LIN {X 0,Y 456.825,Z 300.941,A -85,B 0,C 180,E1 -8385.675,E2 -8385.675} C_VEL
LIN {X 0,Y 457.17,Z 278.124,A -85,B 0,C 180,E1 -8386.064,E2 -8386.064} C_VEL
LIN {X 0,Y 457.468,Z 213.976,A -85,B 0,C 180,E1 -8387.081,E2 -8387.081} C_VEL
LIN {X 0,Y 453.923,Z 193.615,A -85,B 0,C 180,E1 -8387.574,E2 -8387.574} C_VEL
LIN {X 0,Y 453.952,Z 192.33,A -85,B 0,C 180,E1 -8387.805,E2 -8387.805} C_VEL
LIN {X 0,Y 454.571,Z 180.455,A -85,B 0,C 180,E1 -8390.593,E2 -8390.593} C_VEL
LIN {X 0,Y 455.351,Z 165.331,A -85,B 0,C 180,E1 -8394.045,E2 -8394.045} C_VEL
LIN {X 0,Y 455.413,Z 159.694,A -85,B 0,C 180,E1 -8395.356,E2 -8395.356} C_VEL
LIN {X 0,Y 453.574,Z 149.578,A -85,B 0,C 180,E1 -8397.969,E2 -8397.969} C_VEL
LIN {X 0,Y 453.468,Z 149.499,A -85,B 0,C 180,E1 -8401.525,E2 -8401.525} C_VEL
LIN {X 0,Y 453.488,Z 149.492,A -85,B 0,C 180,E1 -8404.777,E2 -8404.777} C_VEL
LIN {X 0,Y 453.474,Z 149.495,A -85,B 0,C 180,E1 -8408.31,E2 -8408.31} C_VEL
LIN {X 0,Y 453.495,Z 149.481,A -85,B 0,C 180,E1 -8410.608,E2 -8410.608} C_VEL
LIN {X 0,Y 453.455,Z 149.501,A -85,B 0,C 180,E1 -8413.243,E2 -8413.243} C_VEL
LIN {X 0,Y 453.461,Z 149.499,A -85,B 0,C 180,E1 -8415.778,E2 -8415.778} C_VEL
LIN {X 0,Y 453.478,Z 149.495,A -85,B 0,C 180,E1 -8418.209,E2 -8418.209} C_VEL
LIN {X 0,Y 453.486,Z 149.489,A -85,B 0,C 180,E1 -8420.794,E2 -8420.794} C_VEL
LIN {X 0,Y 453.453,Z 149.496,A -85,B 0,C 180,E1 -8423.917,E2 -8423.917} C_VEL
LIN {X 0,Y 453.482,Z 149.491,A -85,B 0,C 180,E1 -8427.151,E2 -8427.151} C_VEL
LIN {X 0,Y 453.473,Z 149.494,A -85,B 0,C 180,E1 -8430.268,E2 -8430.268} C_VEL
LIN {X 0,Y 453.504,Z 149.483,A -85,B 0,C 180,E1 -8433.293,E2 -8433.293} C_VEL
LIN {X 0,Y 453.501,Z 149.49,A -85,B 0,C 180,E1 -8436.238,E2 -8436.238} C_VEL
LIN {X 0,Y 453.48,Z 149.49,A -85,B 0,C 180,E1 -8439.117,E2 -8439.117} C_VEL
LIN {X 0,Y 453.509,Z 149.476,A -85,B 0,C 180,E1 -8441.944,E2 -8441.944} C_VEL
LIN {X 0,Y 453.537,Z 149.489,A -85,B 0,C 180,E1 -8444.726,E2 -8444.726} C_VEL
LIN {X 0,Y 453.556,Z 149.483,A -85,B 0,C 180,E1 -8448.378,E2 -8448.378} C_VEL
LIN {X 0,Y 453.649,Z 149.463,A -85,B 0,C 180,E1 -8451.985,E2 -8451.985} C_VEL
LIN {X 0,Y 453.667,Z 149.476,A -85,B 0,C 180,E1 -8454.666,E2 -8454.666} C_VEL
LIN {X 0,Y 453.741,Z 149.457,A -85,B 0,C 180,E1 -8457.336,E2 -8457.336} C_VEL
LIN {X 0,Y 453.819,Z 149.438,A -85,B 0,C 180,E1 -8460,E2 -8460} C_VEL
LIN {X 0,Y 453.761,Z 149.46,A -85,B 0,C 180,E1 -8462.663,E2 -8462.663} C_VEL
LIN {X 0,Y 453.673,Z 149.474,A -85,B 0,C 180,E1 -8466.225,E2 -8466.225} C_VEL
LIN {X 0,Y 453.588,Z 149.467,A -85,B 0,C 180,E1 -8468.913,E2 -8468.913} C_VEL
LIN {X 0,Y 453.559,Z 149.484,A -85,B 0,C 180,E1 -8472.528,E2 -8472.528} C_VEL
LIN {X 0,Y 453.54,Z 149.486,A -85,B 0,C 180,E1 -8476.196,E2 -8476.196} C_VEL
LIN {X 0,Y 453.515,Z 149.473,A -85,B 0,C 180,E1 -8479.04,E2 -8479.04} C_VEL
LIN {X 0,Y 453.472,Z 149.498,A -85,B 0,C 180,E1 -8481.836,E2 -8481.836} C_VEL
LIN {X 0,Y 453.51,Z 149.489,A -85,B 0,C 180,E1 -8484.734,E2 -8484.734} C_VEL
LIN {X 0,Y 453.532,Z 149.483,A -85,B 0,C 180,E1 -8487.961,E2 -8487.961} C_VEL
LIN {X 0,Y 453.476,Z 149.495,A -85,B 0,C 180,E1 -8490.759,E2 -8490.759} C_VEL
LIN {X 0,Y 453.473,Z 149.486,A -85,B 0,C 180,E1 -8493.912,E2 -8493.912} C_VEL
LIN {X 0,Y 453.465,Z 149.5,A -85,B 0,C 180,E1 -8497.188,E2 -8497.188} C_VEL
LIN {X 0,Y 453.5,Z 149.491,A -85,B 0,C 180,E1 -8499.448,E2 -8499.448} C_VEL
LIN {X 0,Y 453.463,Z 149.5,A -85,B 0,C 180,E1 -8502.994,E2 -8502.994} C_VEL
LIN {X 0,Y 453.467,Z 149.487,A -85,B 0,C 180,E1 -8505.78,E2 -8505.78} C_VEL
LIN {X 0,Y 453.489,Z 149.482,A -85,B 0,C 180,E1 -8509.391,E2 -8509.391} C_VEL
LIN {X 0,Y 453.468,Z 149.497,A -85,B 0,C 180,E1 -8512.223,E2 -8512.223} C_VEL
LIN {X 0,Y 453.484,Z 149.481,A -85,B 0,C 180,E1 -8515.222,E2 -8515.222} C_VEL
LIN {X 0,Y 453.483,Z 149.498,A -85,B 0,C 180,E1 -8518.47,E2 -8518.47} C_VEL
LIN {X 0,Y 453.511,Z 149.487,A -85,B 0,C 180,E1 -8521.289,E2 -8521.289} C_VEL
LIN {X 0,Y 453.52,Z 149.494,A -85,B 0,C 180,E1 -8524.285,E2 -8524.285} C_VEL
LIN {X 0,Y 453.476,Z 149.498,A -85,B 0,C 180,E1 -8527.204,E2 -8527.204} C_VEL
LIN {X 0,Y 453.501,Z 149.496,A -85,B 0,C 180,E1 -8530.066,E2 -8530.066} C_VEL
LIN {X 0,Y 453.503,Z 149.497,A -85,B 0,C 180,E1 -8532.876,E2 -8532.876} C_VEL
LIN {X 0,Y 453.51,Z 149.494,A -85,B 0,C 180,E1 -8535.644,E2 -8535.644} C_VEL
LIN {X 0,Y 453.557,Z 149.491,A -85,B 0,C 180,E1 -8538.379,E2 -8538.379} C_VEL
LIN {X 0,Y 453.648,Z 149.479,A -85,B 0,C 180,E1 -8541.985,E2 -8541.985} C_VEL
LIN {X 0,Y 453.633,Z 149.479,A -85,B 0,C 180,E1 -8543.08,E2 -8543.08} C_VEL
LIN {X 0,Y 452.947,Z 149.567,A -85,B 0,C 180,E1 -8543.82,E2 -8543.82} C_VEL
LIN {X 0,Y 449.998,Z 149.932,A -85,B 0,C 180,E1 -8545.022,E2 -8545.022} C_VEL
LIN {X 0,Y 447.574,Z 150.236,A -85,B 0,C 180,E1 -8545.992,E2 -8545.992} C_VEL
LIN {X 0,Y 446.637,Z 150.352,A -85,B 0,C 180,E1 -8546.742,E2 -8546.742} C_VEL
LIN {X 0,Y 446.617,Z 150.352,A -85,B 0,C 180,E1 -8546.995,E2 -8546.995} C_VEL
LIN {X 0,Y 446.791,Z 150.334,A -85,B 0,C 180,E1 -8550,E2 -8550} C_VEL
LIN {X 0,Y 446.706,Z 150.342,A -85,B 0,C 180,E1 -8552.705,E2 -8552.705} C_VEL
LIN {X 0,Y 446.644,Z 150.351,A -85,B 0,C 180,E1 -8556.324,E2 -8556.324} C_VEL
LIN {X 0,Y 446.535,Z 150.364,A -85,B 0,C 180,E1 -8559.055,E2 -8559.055} C_VEL
LIN {X 0,Y 446.517,Z 150.365,A -85,B 0,C 180,E1 -8562.73,E2 -8562.73} C_VEL
LIN {X 0,Y 446.492,Z 150.369,A -85,B 0,C 180,E1 -8566.228,E2 -8566.228} C_VEL
LIN {X 0,Y 446.466,Z 150.375,A -85,B 0,C 180,E1 -8569.303,E2 -8569.303} C_VEL
LIN {X 0,Y 446.415,Z 150.377,A -85,B 0,C 180,E1 -8572.2,E2 -8572.2} C_VEL
LIN {X 0,Y 446.454,Z 150.376,A -85,B 0,C 180,E1 -8575.152,E2 -8575.152} C_VEL
LIN {X 0,Y 446.48,Z 150.365,A -85,B 0,C 180,E1 -8578.179,E2 -8578.179} C_VEL
LIN {X 0,Y 446.43,Z 150.378,A -85,B 0,C 180,E1 -8581.299,E2 -8581.299} C_VEL
LIN {X 0,Y 446.425,Z 150.36,A -85,B 0,C 180,E1 -8584.523,E2 -8584.523} C_VEL
LIN {X 0,Y 446.426,Z 150.374,A -85,B 0,C 180,E1 -8588.082,E2 -8588.082} C_VEL
LIN {X 0,Y 446.421,Z 150.355,A -85,B 0,C 180,E1 -8590.918,E2 -8590.918} C_VEL
LIN {X 0,Y 446.417,Z 150.363,A -85,B 0,C 180,E1 -8593.843,E2 -8593.843} C_VEL
LIN {X 0,Y 446.416,Z 150.377,A -85,B 0,C 180,E1 -8596.4,E2 -8596.4} C_VEL
LIN {X 0,Y 446.443,Z 150.364,A -85,B 0,C 180,E1 -8599.803,E2 -8599.803} C_VEL
LIN {X 0,Y 446.422,Z 150.376,A -85,B 0,C 180,E1 -8602.123,E2 -8602.123} C_VEL
LIN {X 0,Y 446.425,Z 150.361,A -85,B 0,C 180,E1 -8605.477,E2 -8605.477} C_VEL
LIN {X 0,Y 446.413,Z 150.379,A -85,B 0,C 180,E1 -8608.7,E2 -8608.7} C_VEL
LIN {X 0,Y 446.479,Z 150.362,A -85,B 0,C 180,E1 -8611.822,E2 -8611.822} C_VEL
LIN {X 0,Y 446.454,Z 150.369,A -85,B 0,C 180,E1 -8614.848,E2 -8614.848} C_VEL
LIN {X 0,Y 446.443,Z 150.372,A -85,B 0,C 180,E1 -8618.245,E2 -8618.245} C_VEL
LIN {X 0,Y 446.452,Z 150.355,A -85,B 0,C 180,E1 -8621.65,E2 -8621.65} C_VEL
LIN {X 0,Y 446.503,Z 150.365,A -85,B 0,C 180,E1 -8624.48,E2 -8624.48} C_VEL
LIN {X 0,Y 446.513,Z 150.355,A -85,B 0,C 180,E1 -8628.193,E2 -8628.193} C_VEL
LIN {X 0,Y 446.596,Z 150.345,A -85,B 0,C 180,E1 -8631.858,E2 -8631.858} C_VEL
LIN {X 0,Y 446.641,Z 150.346,A -85,B 0,C 180,E1 -8634.583,E2 -8634.583} C_VEL
LIN {X 0,Y 446.705,Z 150.338,A -85,B 0,C 180,E1 -8637.295,E2 -8637.295} C_VEL
LIN {X 0,Y 446.789,Z 150.313,A -85,B 0,C 180,E1 -8640,E2 -8640} C_VEL
LIN {X 0,Y 446.688,Z 150.336,A -85,B 0,C 180,E1 -8642.706,E2 -8642.706} C_VEL
LIN {X 0,Y 446.643,Z 150.343,A -85,B 0,C 180,E1 -8646.324,E2 -8646.324} C_VEL
LIN {X 0,Y 446.534,Z 150.347,A -85,B 0,C 180,E1 -8649.056,E2 -8649.056} C_VEL
LIN {X 0,Y 446.519,Z 150.358,A -85,B 0,C 180,E1 -8652.73,E2 -8652.73} C_VEL
LIN {X 0,Y 446.494,Z 150.359,A -85,B 0,C 180,E1 -8656.228,E2 -8656.228} C_VEL
LIN {X 0,Y 446.467,Z 150.357,A -85,B 0,C 180,E1 -8659.304,E2 -8659.304} C_VEL
LIN {X 0,Y 446.416,Z 150.372,A -85,B 0,C 180,E1 -8662.2,E2 -8662.2} C_VEL
LIN {X 0,Y 446.455,Z 150.365,A -85,B 0,C 180,E1 -8665.153,E2 -8665.153} C_VEL
LIN {X 0,Y 446.483,Z 150.357,A -85,B 0,C 180,E1 -8668.179,E2 -8668.179} C_VEL
LIN {X 0,Y 446.418,Z 150.373,A -85,B 0,C 180,E1 -8671.776,E2 -8671.776} C_VEL
LIN {X 0,Y 446.428,Z 150.366,A -85,B 0,C 180,E1 -8674.524,E2 -8674.524} C_VEL
LIN {X 0,Y 446.412,Z 150.377,A -85,B 0,C 180,E1 -8678.079,E2 -8678.079} C_VEL
LIN {X 0,Y 446.426,Z 150.375,A -85,B 0,C 180,E1 -8680.918,E2 -8680.918} C_VEL
LIN {X 0,Y 446.397,Z 150.377,A -85,B 0,C 180,E1 -8683.847,E2 -8683.847} C_VEL
LIN {X 0,Y 446.398,Z 150.383,A -85,B 0,C 180,E1 -8686.404,E2 -8686.404} C_VEL
LIN {X 0,Y 446.427,Z 150.361,A -85,B 0,C 180,E1 -8689.083,E2 -8689.083} C_VEL
LIN {X 0,Y 446.428,Z 150.377,A -85,B 0,C 180,E1 -8692.124,E2 -8692.124} C_VEL
LIN {X 0,Y 446.43,Z 150.371,A -85,B 0,C 180,E1 -8695.477,E2 -8695.477} C_VEL
LIN {X 0,Y 446.418,Z 150.38,A -85,B 0,C 180,E1 -8698.7,E2 -8698.7} C_VEL
LIN {X 0,Y 446.522,Z 150.503,A -85,B 0,C 180,E1 -8701.824,E2 -8701.824} C_VEL
LIN {X 0,Y 448.185,Z 159.571,A -85,B 0,C 180,E1 -8704.206,E2 -8704.206} C_VEL
LIN {X 0,Y 448.462,Z 164.125,A -85,B 0,C 180,E1 -8705.36,E2 -8705.36} C_VEL
LIN {X 0,Y 447.654,Z 179.053,A -85,B 0,C 180,E1 -8708.833,E2 -8708.833} C_VEL
LIN {X 0,Y 446.966,Z 192.145,A -85,B 0,C 180,E1 -8711.908,E2 -8711.908} C_VEL
LIN {X 0,Y 446.955,Z 193.46,A -85,B 0,C 180,E1 -8712.145,E2 -8712.145} C_VEL
LIN {X 0,Y 450.797,Z 215.824,A -85,B 0,C 180,E1 -8712.691,E2 -8712.691} C_VEL
LIN {X 0,Y 450.061,Z 298.086,A -85,B 0,C 180,E1 -8714.025,E2 -8714.025} C_VEL
LIN {X 0,Y 449.811,Z 307.982,A -85,B 0,C 180,E1 -8714.277,E2 -8714.277} C_VEL
LIN {X 0,Y 449.447,Z 317.957,A -85,B 0,C 180,E1 -8714.642,E2 -8714.642} C_VEL
LIN {X 0,Y 449.065,Z 327.314,A -85,B 0,C 180,E1 -8715.093,E2 -8715.093} C_VEL
LIN {X 0,Y 448.597,Z 335.823,A -85,B 0,C 180,E1 -8715.599,E2 -8715.599} C_VEL
LIN {X 0,Y 448.084,Z 345.1,A -85,B 0,C 180,E1 -8716.277,E2 -8716.277} C_VEL
LIN {X 0,Y 447.67,Z 353.812,A -85,B 0,C 180,E1 -8717.049,E2 -8717.049} C_VEL
LIN {X 0,Y 447.137,Z 362.58,A -85,B 0,C 180,E1 -8717.98,E2 -8717.98} C_VEL
LIN {X 0,Y 446.696,Z 369.8,A -85,B 0,C 180,E1 -8718.888,E2 -8718.888} C_VEL
LIN {X 0,Y 446.358,Z 376.003,A -85,B 0,C 180,E1 -8719.797,E2 -8719.797} C_VEL
LIN {X 0,Y 445.997,Z 382.54,A -85,B 0,C 180,E1 -8720.934,E2 -8720.934} C_VEL
LIN {X 0,Y 445.785,Z 387.041,A -85,B 0,C 180,E1 -8721.843,E2 -8721.843} C_VEL
LIN {X 0,Y 445.57,Z 392.533,A -85,B 0,C 180,E1 -8723.207,E2 -8723.207} C_VEL
LIN {X 0,Y 445.476,Z 396.854,A -85,B 0,C 180,E1 -8724.568,E2 -8724.568} C_VEL
LIN {X 0,Y 445.413,Z 399.219,A -85,B 0,C 180,E1 -8725.475,E2 -8725.475} C_VEL
LIN {X 0,Y 445.433,Z 402.402,A -85,B 0,C 180,E1 -8727.287,E2 -8727.287} C_VEL
LIN {X 0,Y 445.356,Z 403.457,A -85,B 0,C 180,E1 -8728.191,E2 -8728.191} C_VEL
LIN {X 0,Y 445.34,Z 404.044,A -85,B 0,C 180,E1 -8729.096,E2 -8729.096} C_VEL
LIN {X 0,Y 445.34,Z 404.044,A -85,B 0,C 180,E1 -8730.904,E2 -8730.904} C_VEL
LIN {X 0,Y 445.356,Z 403.457,A -85,B 0,C 180,E1 -8731.809,E2 -8731.809} C_VEL
LIN {X 0,Y 445.433,Z 402.402,A -85,B 0,C 180,E1 -8732.713,E2 -8732.713} C_VEL
LIN {X 0,Y 445.413,Z 399.219,A -85,B 0,C 180,E1 -8734.525,E2 -8734.525} C_VEL
LIN {X 0,Y 445.469,Z 395.105,A -85,B 0,C 180,E1 -8736.041,E2 -8736.041} C_VEL
LIN {X 0,Y 445.601,Z 390.871,A -85,B 0,C 180,E1 -8737.249,E2 -8737.249} C_VEL
LIN {X 0,Y 445.889,Z 384.851,A -85,B 0,C 180,E1 -8738.612,E2 -8738.612} C_VEL
LIN {X 0,Y 446.194,Z 378.755,A -85,B 0,C 180,E1 -8739.748,E2 -8739.748} C_VEL
LIN {X 0,Y 446.498,Z 373.054,A -85,B 0,C 180,E1 -8740.658,E2 -8740.658} C_VEL
LIN {X 0,Y 447.04,Z 364.5,A -85,B 0,C 180,E1 -8741.793,E2 -8741.793} C_VEL
LIN {X 0,Y 447.502,Z 356.319,A -85,B 0,C 180,E1 -8742.701,E2 -8742.701} C_VEL
LIN {X 0,Y 447.957,Z 347.932,A -85,B 0,C 180,E1 -8743.485,E2 -8743.485} C_VEL
LIN {X 0,Y 448.42,Z 339.087,A -85,B 0,C 180,E1 -8744.175,E2 -8744.175} C_VEL
LIN {X 0,Y 448.916,Z 329.327,A -85,B 0,C 180,E1 -8744.796,E2 -8744.796} C_VEL
LIN {X 0,Y 449.344,Z 320.533,A -85,B 0,C 180,E1 -8745.245,E2 -8745.245} C_VEL
LIN {X 0,Y 449.727,Z 310.605,A -85,B 0,C 180,E1 -8745.639,E2 -8745.639} C_VEL
LIN {X 0,Y 450.008,Z 300.75,A -85,B 0,C 180,E1 -8745.919,E2 -8745.919} C_VEL
LIN {X 0,Y 450.402,Z 275.651,A -85,B 0,C 180,E1 -8746.349,E2 -8746.349} C_VEL
LIN {X 0,Y 450.678,Z 214.695,A -85,B 0,C 180,E1 -8747.332,E2 -8747.332} C_VEL
LIN {X 0,Y 446.964,Z 193.579,A -85,B 0,C 180,E1 -8747.846,E2 -8747.846} C_VEL
LIN {X 0,Y 446.931,Z 192.787,A -85,B 0,C 180,E1 -8747.942,E2 -8747.942} C_VEL
LIN {X 0,Y 447.636,Z 180.293,A -85,B 0,C 180,E1 -8750.927,E2 -8750.927} C_VEL
LIN {X 0,Y 448.451,Z 165.578,A -85,B 0,C 180,E1 -8754.349,E2 -8754.349} C_VEL
LIN {X 0,Y 448.395,Z 160.582,A -85,B 0,C 180,E1 -8755.532,E2 -8755.532} C_VEL
LIN {X 0,Y 446.524,Z 150.482,A -85,B 0,C 180,E1 -8758.187,E2 -8758.187} C_VEL
LIN {X 0,Y 446.421,Z 150.374,A -85,B 0,C 180,E1 -8761.774,E2 -8761.774} C_VEL
LIN {X 0,Y 446.43,Z 150.372,A -85,B 0,C 180,E1 -8764.523,E2 -8764.523} C_VEL
LIN {X 0,Y 446.431,Z 150.375,A -85,B 0,C 180,E1 -8768.081,E2 -8768.081} C_VEL
LIN {X 0,Y 446.427,Z 150.361,A -85,B 0,C 180,E1 -8770.917,E2 -8770.917} C_VEL
LIN {X 0,Y 446.4,Z 150.379,A -85,B 0,C 180,E1 -8773.846,E2 -8773.846} C_VEL
LIN {X 0,Y 446.396,Z 150.377,A -85,B 0,C 180,E1 -8776.403,E2 -8776.403} C_VEL
LIN {X 0,Y 446.426,Z 150.375,A -85,B 0,C 180,E1 -8779.082,E2 -8779.082} C_VEL
LIN {X 0,Y 446.406,Z 150.376,A -85,B 0,C 180,E1 -8782.12,E2 -8782.12} C_VEL
LIN {X 0,Y 446.428,Z 150.366,A -85,B 0,C 180,E1 -8785.476,E2 -8785.476} C_VEL
LIN {X 0,Y 446.415,Z 150.375,A -85,B 0,C 180,E1 -8788.699,E2 -8788.699} C_VEL
LIN {X 0,Y 446.483,Z 150.357,A -85,B 0,C 180,E1 -8791.821,E2 -8791.821} C_VEL
LIN {X 0,Y 446.455,Z 150.365,A -85,B 0,C 180,E1 -8794.847,E2 -8794.847} C_VEL
LIN {X 0,Y 446.446,Z 150.369,A -85,B 0,C 180,E1 -8798.245,E2 -8798.245} C_VEL
LIN {X 0,Y 446.454,Z 150.354,A -85,B 0,C 180,E1 -8801.649,E2 -8801.649} C_VEL
LIN {X 0,Y 446.505,Z 150.362,A -85,B 0,C 180,E1 -8804.479,E2 -8804.479} C_VEL
LIN {X 0,Y 446.514,Z 150.359,A -85,B 0,C 180,E1 -8808.193,E2 -8808.193} C_VEL
LIN {X 0,Y 446.597,Z 150.34,A -85,B 0,C 180,E1 -8811.857,E2 -8811.857} C_VEL
LIN {X 0,Y 446.642,Z 150.352,A -85,B 0,C 180,E1 -8814.582,E2 -8814.582} C_VEL
LIN {X 0,Y 446.66,Z 150.34,A -85,B 0,C 180,E1 -8818.196,E2 -8818.196} C_VEL
LIN {X 0,Y 446.789,Z 150.313,A -85,B 0,C 180,E1 -8820,E2 -8820} C_VEL
LIN {X 0,Y 446.705,Z 150.338,A -85,B 0,C 180,E1 -8822.705,E2 -8822.705} C_VEL
LIN {X 0,Y 446.642,Z 150.348,A -85,B 0,C 180,E1 -8826.323,E2 -8826.323} C_VEL
LIN {X 0,Y 446.534,Z 150.344,A -85,B 0,C 180,E1 -8829.055,E2 -8829.055} C_VEL
LIN {X 0,Y 446.517,Z 150.36,A -85,B 0,C 180,E1 -8832.729,E2 -8832.729} C_VEL
LIN {X 0,Y 446.492,Z 150.364,A -85,B 0,C 180,E1 -8836.228,E2 -8836.228} C_VEL
LIN {X 0,Y 446.464,Z 150.352,A -85,B 0,C 180,E1 -8839.303,E2 -8839.303} C_VEL
LIN {X 0,Y 446.414,Z 150.377,A -85,B 0,C 180,E1 -8842.199,E2 -8842.199} C_VEL
LIN {X 0,Y 446.454,Z 150.369,A -85,B 0,C 180,E1 -8845.152,E2 -8845.152} C_VEL
LIN {X 0,Y 446.479,Z 150.362,A -85,B 0,C 180,E1 -8848.178,E2 -8848.178} C_VEL
LIN {X 0,Y 446.413,Z 150.379,A -85,B 0,C 180,E1 -8851.3,E2 -8851.3} C_VEL
LIN {X 0,Y 446.425,Z 150.361,A -85,B 0,C 180,E1 -8854.523,E2 -8854.523} C_VEL
LIN {X 0,Y 446.425,Z 150.374,A -85,B 0,C 180,E1 -8858.082,E2 -8858.082} C_VEL
LIN {X 0,Y 446.422,Z 150.368,A -85,B 0,C 180,E1 -8860.918,E2 -8860.918} C_VEL
LIN {X 0,Y 446.418,Z 150.374,A -85,B 0,C 180,E1 -8863.843,E2 -8863.843} C_VEL
LIN {X 0,Y 446.415,Z 150.364,A -85,B 0,C 180,E1 -8866.4,E2 -8866.4} C_VEL
LIN {X 0,Y 446.438,Z 150.366,A -85,B 0,C 180,E1 -8869.802,E2 -8869.802} C_VEL
LIN {X 0,Y 446.423,Z 150.375,A -85,B 0,C 180,E1 -8872.123,E2 -8872.123} C_VEL
LIN {X 0,Y 446.426,Z 150.36,A -85,B 0,C 180,E1 -8875.477,E2 -8875.477} C_VEL
LIN {X 0,Y 446.43,Z 150.378,A -85,B 0,C 180,E1 -8878.701,E2 -8878.701} C_VEL
LIN {X 0,Y 446.48,Z 150.365,A -85,B 0,C 180,E1 -8881.821,E2 -8881.821} C_VEL
LIN {X 0,Y 446.454,Z 150.376,A -85,B 0,C 180,E1 -8884.848,E2 -8884.848} C_VEL
LIN {X 0,Y 446.444,Z 150.376,A -85,B 0,C 180,E1 -8888.245,E2 -8888.245} C_VEL
LIN {X 0,Y 446.454,Z 150.373,A -85,B 0,C 180,E1 -8891.649,E2 -8891.649} C_VEL
LIN {X 0,Y 446.504,Z 150.37,A -85,B 0,C 180,E1 -8894.48,E2 -8894.48} C_VEL
LIN {X 0,Y 446.514,Z 150.368,A -85,B 0,C 180,E1 -8898.193,E2 -8898.193} C_VEL
LIN {X 0,Y 446.597,Z 150.357,A -85,B 0,C 180,E1 -8901.858,E2 -8901.858} C_VEL
LIN {X 0,Y 446.643,Z 150.351,A -85,B 0,C 180,E1 -8904.583,E2 -8904.583} C_VEL
LIN {X 0,Y 446.617,Z 150.352,A -85,B 0,C 180,E1 -8906.995,E2 -8906.995} C_VEL
LIN {X 0,Y 446.1,Z 150.42,A -85,B 0,C 180,E1 -8907.748,E2 -8907.748} C_VEL
LIN {X 0,Y 443.286,Z 150.772,A -85,B 0,C 180,E1 -8908.971,E2 -8908.971} C_VEL
LIN {X 0,Y 440.802,Z 151.081,A -85,B 0,C 180,E1 -8909.958,E2 -8909.958} C_VEL
LIN {X 0,Y 439.713,Z 151.214,A -85,B 0,C 180,E1 -8910.721,E2 -8910.721} C_VEL
LIN {X 0,Y 439.619,Z 151.225,A -85,B 0,C 180,E1 -8910.98,E2 -8910.98} C_VEL
LIN {X 0,Y 439.653,Z 151.221,A -85,B 0,C 180,E1 -8912.749,E2 -8912.749} C_VEL
LIN {X 0,Y 439.615,Z 151.226,A -85,B 0,C 180,E1 -8916.425,E2 -8916.425} C_VEL
LIN {X 0,Y 439.497,Z 151.241,A -85,B 0,C 180,E1 -8919.202,E2 -8919.202} C_VEL
LIN {X 0,Y 439.462,Z 151.245,A -85,B 0,C 180,E1 -8922.938,E2 -8922.938} C_VEL
LIN {X 0,Y 439.444,Z 151.246,A -85,B 0,C 180,E1 -8926.349,E2 -8926.349} C_VEL
LIN {X 0,Y 439.399,Z 151.255,A -85,B 0,C 180,E1 -8929.626,E2 -8929.626} C_VEL
LIN {X 0,Y 439.362,Z 151.256,A -85,B 0,C 180,E1 -8932.575,E2 -8932.575} C_VEL
LIN {X 0,Y 439.401,Z 151.254,A -85,B 0,C 180,E1 -8935.585,E2 -8935.585} C_VEL
LIN {X 0,Y 439.421,Z 151.241,A -85,B 0,C 180,E1 -8938.673,E2 -8938.673} C_VEL
LIN {X 0,Y 439.381,Z 151.252,A -85,B 0,C 180,E1 -8942.034,E2 -8942.034} C_VEL
LIN {X 0,Y 439.391,Z 151.239,A -85,B 0,C 180,E1 -8945.341,E2 -8945.341} C_VEL
LIN {X 0,Y 439.379,Z 151.255,A -85,B 0,C 180,E1 -8948.595,E2 -8948.595} C_VEL
LIN {X 0,Y 439.383,Z 151.226,A -85,B 0,C 180,E1 -8951.257,E2 -8951.257} C_VEL
LIN {X 0,Y 439.401,Z 151.243,A -85,B 0,C 180,E1 -8954.729,E2 -8954.729} C_VEL
LIN {X 0,Y 439.393,Z 151.248,A -85,B 0,C 180,E1 -8957.796,E2 -8957.796} C_VEL
LIN {X 0,Y 439.425,Z 151.24,A -85,B 0,C 180,E1 -8960.228,E2 -8960.228} C_VEL
LIN {X 0,Y 439.372,Z 151.251,A -85,B 0,C 180,E1 -8963.713,E2 -8963.713} C_VEL
LIN {X 0,Y 439.368,Z 151.252,A -85,B 0,C 180,E1 -8967.054,E2 -8967.054} C_VEL
LIN {X 0,Y 439.386,Z 151.254,A -85,B 0,C 180,E1 -8970.275,E2 -8970.275} C_VEL
LIN {X 0,Y 439.425,Z 151.234,A -85,B 0,C 180,E1 -8973.397,E2 -8973.397} C_VEL
LIN {X 0,Y 439.383,Z 151.255,A -85,B 0,C 180,E1 -8976.43,E2 -8976.43} C_VEL
LIN {X 0,Y 439.383,Z 151.244,A -85,B 0,C 180,E1 -8979.397,E2 -8979.397} C_VEL
LIN {X 0,Y 439.427,Z 151.239,A -85,B 0,C 180,E1 -8982.31,E2 -8982.31} C_VEL
LIN {X 0,Y 439.443,Z 151.243,A -85,B 0,C 180,E1 -8985.174,E2 -8985.174} C_VEL
LIN {X 0,Y 439.479,Z 151.233,A -85,B 0,C 180,E1 -8988.002,E2 -8988.002} C_VEL
LIN {X 0,Y 439.544,Z 151.221,A -85,B 0,C 180,E1 -8991.727,E2 -8991.727} C_VEL
LIN {X 0,Y 439.617,Z 151.221,A -85,B 0,C 180,E1 -8994.496,E2 -8994.496} C_VEL
LIN {X 0,Y 439.632,Z 151.208,A -85,B 0,C 180,E1 -8998.168,E2 -8998.168} C_VEL
LIN {X 0,Y 439.758,Z 151.188,A -85,B 0,C 180,E1 -9000,E2 -9000} C_VEL
LIN {X 0,Y 439.638,Z 151.214,A -85,B 0,C 180,E1 -9002.749,E2 -9002.749} C_VEL
LIN {X 0,Y 439.615,Z 151.219,A -85,B 0,C 180,E1 -9006.426,E2 -9006.426} C_VEL
LIN {X 0,Y 439.496,Z 151.222,A -85,B 0,C 180,E1 -9009.202,E2 -9009.202} C_VEL
LIN {X 0,Y 439.463,Z 151.238,A -85,B 0,C 180,E1 -9012.938,E2 -9012.938} C_VEL
LIN {X 0,Y 439.445,Z 151.238,A -85,B 0,C 180,E1 -9016.349,E2 -9016.349} C_VEL
LIN {X 0,Y 439.4,Z 151.24,A -85,B 0,C 180,E1 -9019.627,E2 -9019.627} C_VEL
LIN {X 0,Y 439.363,Z 151.253,A -85,B 0,C 180,E1 -9022.576,E2 -9022.576} C_VEL
LIN {X 0,Y 439.403,Z 151.239,A -85,B 0,C 180,E1 -9025.585,E2 -9025.585} C_VEL
LIN {X 0,Y 439.416,Z 151.242,A -85,B 0,C 180,E1 -9028.674,E2 -9028.674} C_VEL
LIN {X 0,Y 439.369,Z 151.251,A -85,B 0,C 180,E1 -9032.031,E2 -9032.031} C_VEL
LIN {X 0,Y 439.393,Z 151.246,A -85,B 0,C 180,E1 -9035.341,E2 -9035.341} C_VEL
LIN {X 0,Y 439.374,Z 151.253,A -85,B 0,C 180,E1 -9038.596,E2 -9038.596} C_VEL
LIN {X 0,Y 439.388,Z 151.249,A -85,B 0,C 180,E1 -9041.257,E2 -9041.257} C_VEL
LIN {X 0,Y 439.399,Z 151.249,A -85,B 0,C 180,E1 -9044.73,E2 -9044.73} C_VEL
LIN {X 0,Y 439.396,Z 151.25,A -85,B 0,C 180,E1 -9047.796,E2 -9047.796} C_VEL
LIN {X 0,Y 439.43,Z 151.234,A -85,B 0,C 180,E1 -9050.228,E2 -9050.228} C_VEL
LIN {X 0,Y 439.375,Z 151.251,A -85,B 0,C 180,E1 -9053.713,E2 -9053.713} C_VEL
LIN {X 0,Y 439.374,Z 151.252,A -85,B 0,C 180,E1 -9057.055,E2 -9057.055} C_VEL
LIN {X 0,Y 439.384,Z 151.25,A -85,B 0,C 180,E1 -9060.275,E2 -9060.275} C_VEL
LIN {X 0,Y 439.476,Z 151.376,A -85,B 0,C 180,E1 -9061.589,E2 -9061.589} C_VEL
LIN {X 0,Y 441.152,Z 160.441,A -85,B 0,C 180,E1 -9064.017,E2 -9064.017} C_VEL
LIN {X 0,Y 441.533,Z 164.726,A -85,B 0,C 180,E1 -9065.133,E2 -9065.133} C_VEL
LIN {X 0,Y 440.669,Z 179.922,A -85,B 0,C 180,E1 -9068.726,E2 -9068.726} C_VEL
LIN {X 0,Y 439.998,Z 191.956,A -85,B 0,C 180,E1 -9071.612,E2 -9071.612} C_VEL
LIN {X 0,Y 439.991,Z 193.272,A -85,B 0,C 180,E1 -9071.853,E2 -9071.853} C_VEL
LIN {X 0,Y 444.019,Z 216.881,A -85,B 0,C 180,E1 -9072.439,E2 -9072.439} C_VEL
LIN {X 0,Y 443.239,Z 297.895,A -85,B 0,C 180,E1 -9073.772,E2 -9073.772} C_VEL
LIN {X 0,Y 442.974,Z 307.79,A -85,B 0,C 180,E1 -9074.028,E2 -9074.028} C_VEL
LIN {X 0,Y 442.615,Z 317.766,A -85,B 0,C 180,E1 -9074.399,E2 -9074.399} C_VEL
LIN {X 0,Y 442.152,Z 328.13,A -85,B 0,C 180,E1 -9074.913,E2 -9074.913} C_VEL
LIN {X 0,Y 441.617,Z 337.263,A -85,B 0,C 180,E1 -9075.484,E2 -9075.484} C_VEL
LIN {X 0,Y 441.101,Z 346.261,A -85,B 0,C 180,E1 -9076.173,E2 -9076.173} C_VEL
LIN {X 0,Y 440.676,Z 354.409,A -85,B 0,C 180,E1 -9076.921,E2 -9076.921} C_VEL
LIN {X 0,Y 440.177,Z 362.388,A -85,B 0,C 180,E1 -9077.787,E2 -9077.787} C_VEL
LIN {X 0,Y 439.712,Z 369.608,A -85,B 0,C 180,E1 -9078.709,E2 -9078.709} C_VEL
LIN {X 0,Y 439.342,Z 375.81,A -85,B 0,C 180,E1 -9079.633,E2 -9079.633} C_VEL
LIN {X 0,Y 438.97,Z 382.348,A -85,B 0,C 180,E1 -9080.787,E2 -9080.787} C_VEL
LIN {X 0,Y 438.739,Z 386.849,A -85,B 0,C 180,E1 -9081.711,E2 -9081.711} C_VEL
LIN {X 0,Y 438.499,Z 392.339,A -85,B 0,C 180,E1 -9083.096,E2 -9083.096} C_VEL
LIN {X 0,Y 438.374,Z 396.662,A -85,B 0,C 180,E1 -9084.48,E2 -9084.48} C_VEL
LIN {X 0,Y 438.342,Z 399.027,A -85,B 0,C 180,E1 -9085.402,E2 -9085.402} C_VEL
LIN {X 0,Y 438.341,Z 402.211,A -85,B 0,C 180,E1 -9087.243,E2 -9087.243} C_VEL
LIN {X 0,Y 438.279,Z 403.266,A -85,B 0,C 180,E1 -9088.162,E2 -9088.162} C_VEL
LIN {X 0,Y 438.253,Z 403.853,A -85,B 0,C 180,E1 -9089.081,E2 -9089.081} C_VEL
LIN {X 0,Y 438.253,Z 403.853,A -85,B 0,C 180,E1 -9090.919,E2 -9090.919} C_VEL
LIN {X 0,Y 438.279,Z 403.266,A -85,B 0,C 180,E1 -9091.838,E2 -9091.838} C_VEL
LIN {X 0,Y 438.341,Z 402.211,A -85,B 0,C 180,E1 -9092.757,E2 -9092.757} C_VEL
LIN {X 0,Y 438.342,Z 399.027,A -85,B 0,C 180,E1 -9094.598,E2 -9094.598} C_VEL
LIN {X 0,Y 438.423,Z 394.227,A -85,B 0,C 180,E1 -9096.343,E2 -9096.343} C_VEL
LIN {X 0,Y 438.633,Z 388.764,A -85,B 0,C 180,E1 -9097.827,E2 -9097.827} C_VEL
LIN {X 0,Y 438.891,Z 383.503,A -85,B 0,C 180,E1 -9098.982,E2 -9098.982} C_VEL
LIN {X 0,Y 439.247,Z 377.186,A -85,B 0,C 180,E1 -9100.137,E2 -9100.137} C_VEL
LIN {X 0,Y 439.582,Z 371.234,A -85,B 0,C 180,E1 -9101.061,E2 -9101.061} C_VEL
LIN {X 0,Y 440.063,Z 364.307,A -85,B 0,C 180,E1 -9101.983,E2 -9101.983} C_VEL
LIN {X 0,Y 440.54,Z 356.126,A -85,B 0,C 180,E1 -9102.905,E2 -9102.905} C_VEL
LIN {X 0,Y 441.009,Z 348.189,A -85,B 0,C 180,E1 -9103.662,E2 -9103.662} C_VEL
LIN {X 0,Y 441.532,Z 338.895,A -85,B 0,C 180,E1 -9104.401,E2 -9104.401} C_VEL
LIN {X 0,Y 442.041,Z 329.135,A -85,B 0,C 180,E1 -9105.031,E2 -9105.031} C_VEL
LIN {X 0,Y 442.599,Z 319.055,A -85,B 0,C 180,E1 -9105.543,E2 -9105.543} C_VEL
LIN {X 0,Y 442.921,Z 309.539,A -85,B 0,C 180,E1 -9105.915,E2 -9105.915} C_VEL
LIN {X 0,Y 443.2,Z 300.559,A -85,B 0,C 180,E1 -9106.17,E2 -9106.17} C_VEL
LIN {X 0,Y 443.601,Z 275.568,A -85,B 0,C 180,E1 -9106.605,E2 -9106.605} C_VEL
LIN {X 0,Y 443.964,Z 215.957,A -85,B 0,C 180,E1 -9107.578,E2 -9107.578} C_VEL
LIN {X 0,Y 439.969,Z 193.239,A -85,B 0,C 180,E1 -9108.15,E2 -9108.15} C_VEL
LIN {X 0,Y 439.983,Z 192.049,A -85,B 0,C 180,E1 -9108.365,E2 -9108.365} C_VEL
LIN {X 0,Y 440.674,Z 180.13,A -85,B 0,C 180,E1 -9111.273,E2 -9111.273} C_VEL
LIN {X 0,Y 441.489,Z 166.736,A -85,B 0,C 180,E1 -9114.449,E2 -9114.449} C_VEL
LIN {X 0,Y 441.527,Z 162.54,A -85,B 0,C 180,E1 -9115.453,E2 -9115.453} C_VEL
LIN {X 0,Y 439.75,Z 152.83,A -85,B 0,C 180,E1 -9118.001,E2 -9118.001} C_VEL
LIN {X 0,Y 439.446,Z 151.268,A -85,B 0,C 180,E1 -9118.493,E2 -9118.493} C_VEL
LIN {X 0,Y 439.372,Z 151.251,A -85,B 0,C 180,E1 -9122.03,E2 -9122.03} C_VEL
LIN {X 0,Y 439.395,Z 151.244,A -85,B 0,C 180,E1 -9125.34,E2 -9125.34} C_VEL
LIN {X 0,Y 439.389,Z 151.248,A -85,B 0,C 180,E1 -9128.594,E2 -9128.594} C_VEL
LIN {X 0,Y 439.389,Z 151.24,A -85,B 0,C 180,E1 -9131.256,E2 -9131.256} C_VEL
LIN {X 0,Y 439.399,Z 151.247,A -85,B 0,C 180,E1 -9134.729,E2 -9134.729} C_VEL
LIN {X 0,Y 439.395,Z 151.252,A -85,B 0,C 180,E1 -9137.795,E2 -9137.795} C_VEL
LIN {X 0,Y 439.394,Z 151.243,A -85,B 0,C 180,E1 -9140.223,E2 -9140.223} C_VEL
LIN {X 0,Y 439.373,Z 151.251,A -85,B 0,C 180,E1 -9143.712,E2 -9143.712} C_VEL
LIN {X 0,Y 439.371,Z 151.247,A -85,B 0,C 180,E1 -9147.053,E2 -9147.053} C_VEL
LIN {X 0,Y 439.381,Z 151.25,A -85,B 0,C 180,E1 -9150.274,E2 -9150.274} C_VEL
LIN {X 0,Y 439.427,Z 151.236,A -85,B 0,C 180,E1 -9153.396,E2 -9153.396} C_VEL
LIN {X 0,Y 439.384,Z 151.249,A -85,B 0,C 180,E1 -9156.429,E2 -9156.429} C_VEL
LIN {X 0,Y 439.386,Z 151.242,A -85,B 0,C 180,E1 -9159.396,E2 -9159.396} C_VEL
LIN {X 0,Y 439.429,Z 151.23,A -85,B 0,C 180,E1 -9162.309,E2 -9162.309} C_VEL
LIN {X 0,Y 439.446,Z 151.244,A -85,B 0,C 180,E1 -9165.173,E2 -9165.173} C_VEL
LIN {X 0,Y 439.48,Z 151.233,A -85,B 0,C 180,E1 -9168.001,E2 -9168.001} C_VEL
LIN {X 0,Y 439.545,Z 151.218,A -85,B 0,C 180,E1 -9171.726,E2 -9171.726} C_VEL
LIN {X 0,Y 439.618,Z 151.226,A -85,B 0,C 180,E1 -9174.495,E2 -9174.495} C_VEL
LIN {X 0,Y 439.63,Z 151.216,A -85,B 0,C 180,E1 -9178.167,E2 -9178.167} C_VEL
LIN {X 0,Y 439.758,Z 151.188,A -85,B 0,C 180,E1 -9180,E2 -9180} C_VEL
LIN {X 0,Y 439.652,Z 151.216,A -85,B 0,C 180,E1 -9182.748,E2 -9182.748} C_VEL
LIN {X 0,Y 439.614,Z 151.222,A -85,B 0,C 180,E1 -9186.425,E2 -9186.425} C_VEL
LIN {X 0,Y 439.496,Z 151.221,A -85,B 0,C 180,E1 -9189.201,E2 -9189.201} C_VEL
LIN {X 0,Y 439.461,Z 151.238,A -85,B 0,C 180,E1 -9192.937,E2 -9192.937} C_VEL
LIN {X 0,Y 439.443,Z 151.24,A -85,B 0,C 180,E1 -9196.348,E2 -9196.348} C_VEL
LIN {X 0,Y 439.398,Z 151.234,A -85,B 0,C 180,E1 -9199.626,E2 -9199.626} C_VEL
LIN {X 0,Y 439.361,Z 151.253,A -85,B 0,C 180,E1 -9202.575,E2 -9202.575} C_VEL
LIN {X 0,Y 439.401,Z 151.246,A -85,B 0,C 180,E1 -9205.584,E2 -9205.584} C_VEL
LIN {X 0,Y 439.416,Z 151.24,A -85,B 0,C 180,E1 -9208.673,E2 -9208.673} C_VEL
LIN {X 0,Y 439.369,Z 151.254,A -85,B 0,C 180,E1 -9211.86,E2 -9211.86} C_VEL
LIN {X 0,Y 439.396,Z 151.24,A -85,B 0,C 180,E1 -9215.156,E2 -9215.156} C_VEL
LIN {X 0,Y 439.383,Z 151.251,A -85,B 0,C 180,E1 -9218.594,E2 -9218.594} C_VEL
LIN {X 0,Y 439.384,Z 151.247,A -85,B 0,C 180,E1 -9221.257,E2 -9221.257} C_VEL
LIN {X 0,Y 439.401,Z 151.25,A -85,B 0,C 180,E1 -9224.728,E2 -9224.728} C_VEL
LIN {X 0,Y 439.391,Z 151.221,A -85,B 0,C 180,E1 -9227.796,E2 -9227.796} C_VEL
LIN {X 0,Y 439.421,Z 151.24,A -85,B 0,C 180,E1 -9230.227,E2 -9230.227} C_VEL
LIN {X 0,Y 439.372,Z 151.247,A -85,B 0,C 180,E1 -9233.713,E2 -9233.713} C_VEL
LIN {X 0,Y 439.372,Z 151.251,A -85,B 0,C 180,E1 -9237.054,E2 -9237.054} C_VEL
LIN {X 0,Y 439.393,Z 151.243,A -85,B 0,C 180,E1 -9240.275,E2 -9240.275} C_VEL
LIN {X 0,Y 439.429,Z 151.247,A -85,B 0,C 180,E1 -9243.589,E2 -9243.589} C_VEL
LIN {X 0,Y 439.383,Z 151.257,A -85,B 0,C 180,E1 -9246.43,E2 -9246.43} C_VEL
LIN {X 0,Y 439.385,Z 151.253,A -85,B 0,C 180,E1 -9249.397,E2 -9249.397} C_VEL
LIN {X 0,Y 439.428,Z 151.251,A -85,B 0,C 180,E1 -9252.31,E2 -9252.31} C_VEL
LIN {X 0,Y 439.444,Z 151.247,A -85,B 0,C 180,E1 -9255.174,E2 -9255.174} C_VEL
LIN {X 0,Y 439.48,Z 151.244,A -85,B 0,C 180,E1 -9258.001,E2 -9258.001} C_VEL
LIN {X 0,Y 439.544,Z 151.236,A -85,B 0,C 180,E1 -9261.726,E2 -9261.726} C_VEL
LIN {X 0,Y 439.618,Z 151.227,A -85,B 0,C 180,E1 -9264.496,E2 -9264.496} C_VEL
LIN {X 0,Y 439.633,Z 151.225,A -85,B 0,C 180,E1 -9268.168,E2 -9268.168} C_VEL
LIN {X 0,Y 439.761,Z 151.21,A -85,B 0,C 180,E1 -9270,E2 -9270} C_VEL
LIN {X 0,Y 439.619,Z 151.225,A -85,B 0,C 180,E1 -9270.98,E2 -9270.98} C_VEL
LIN {X 0,Y 438.902,Z 151.316,A -85,B 0,C 180,E1 -9271.744,E2 -9271.744} C_VEL
LIN {X 0,Y 435.923,Z 151.686,A -85,B 0,C 180,E1 -9272.984,E2 -9272.984} C_VEL
LIN {X 0,Y 433.471,Z 151.993,A -85,B 0,C 180,E1 -9273.984,E2 -9273.984} C_VEL
LIN {X 0,Y 432.497,Z 152.113,A -85,B 0,C 180,E1 -9274.758,E2 -9274.758} C_VEL
LIN {X 0,Y 432.46,Z 152.117,A -85,B 0,C 180,E1 -9275.02,E2 -9275.02} C_VEL
LIN {X 0,Y 432.582,Z 152.103,A -85,B 0,C 180,E1 -9277.679,E2 -9277.679} C_VEL
LIN {X 0,Y 432.39,Z 152.127,A -85,B 0,C 180,E1 -9281.247,E2 -9281.247} C_VEL
LIN {X 0,Y 432.37,Z 152.129,A -85,B 0,C 180,E1 -9284.112,E2 -9284.112} C_VEL
LIN {X 0,Y 432.393,Z 152.126,A -85,B 0,C 180,E1 -9287.011,E2 -9287.011} C_VEL
LIN {X 0,Y 432.335,Z 152.133,A -85,B 0,C 180,E1 -9289.96,E2 -9289.96} C_VEL
LIN {X 0,Y 432.316,Z 152.136,A -85,B 0,C 180,E1 -9292.964,E2 -9292.964} C_VEL
LIN {X 0,Y 432.36,Z 152.128,A -85,B 0,C 180,E1 -9296.032,E2 -9296.032} C_VEL
LIN {X 0,Y 432.348,Z 152.118,A -85,B 0,C 180,E1 -9299.187,E2 -9299.187} C_VEL
LIN {X 0,Y 432.328,Z 152.131,A -85,B 0,C 180,E1 -9302.295,E2 -9302.295} C_VEL
LIN {X 0,Y 432.336,Z 152.113,A -85,B 0,C 180,E1 -9304.677,E2 -9304.677} C_VEL
LIN {X 0,Y 432.34,Z 152.129,A -85,B 0,C 180,E1 -9308.149,E2 -9308.149} C_VEL
LIN {X 0,Y 432.327,Z 152.102,A -85,B 0,C 180,E1 -9311.602,E2 -9311.602} C_VEL
LIN {X 0,Y 432.335,Z 152.119,A -85,B 0,C 180,E1 -9314.347,E2 -9314.347} C_VEL
LIN {X 0,Y 432.32,Z 152.133,A -85,B 0,C 180,E1 -9317.015,E2 -9317.015} C_VEL
LIN {X 0,Y 432.331,Z 152.121,A -85,B 0,C 180,E1 -9319.82,E2 -9319.82} C_VEL
LIN {X 0,Y 432.31,Z 152.133,A -85,B 0,C 180,E1 -9323.023,E2 -9323.023} C_VEL
LIN {X 0,Y 432.354,Z 152.115,A -85,B 0,C 180,E1 -9325.997,E2 -9325.997} C_VEL
LIN {X 0,Y 432.387,Z 152.123,A -85,B 0,C 180,E1 -9329.744,E2 -9329.744} C_VEL
LIN {X 0,Y 432.395,Z 152.109,A -85,B 0,C 180,E1 -9333.373,E2 -9333.373} C_VEL
LIN {X 0,Y 432.367,Z 152.127,A -85,B 0,C 180,E1 -9336.024,E2 -9336.024} C_VEL
LIN {X 0,Y 432.345,Z 152.12,A -85,B 0,C 180,E1 -9339.046,E2 -9339.046} C_VEL
LIN {X 0,Y 432.373,Z 152.111,A -85,B 0,C 180,E1 -9342.012,E2 -9342.012} C_VEL
LIN {X 0,Y 432.391,Z 152.121,A -85,B 0,C 180,E1 -9344.927,E2 -9344.927} C_VEL
LIN {X 0,Y 432.455,Z 152.111,A -85,B 0,C 180,E1 -9347.804,E2 -9347.804} C_VEL
LIN {X 0,Y 432.488,Z 152.097,A -85,B 0,C 180,E1 -9351.591,E2 -9351.591} C_VEL
LIN {X 0,Y 432.594,Z 152.097,A -85,B 0,C 180,E1 -9354.407,E2 -9354.407} C_VEL
LIN {X 0,Y 432.602,Z 152.083,A -85,B 0,C 180,E1 -9358.139,E2 -9358.139} C_VEL
LIN {X 0,Y 432.728,Z 152.062,A -85,B 0,C 180,E1 -9360.001,E2 -9360.001} C_VEL
LIN {X 0,Y 432.59,Z 152.092,A -85,B 0,C 180,E1 -9362.794,E2 -9362.794} C_VEL
LIN {X 0,Y 432.569,Z 152.096,A -85,B 0,C 180,E1 -9366.531,E2 -9366.531} C_VEL
LIN {X 0,Y 432.439,Z 152.099,A -85,B 0,C 180,E1 -9369.354,E2 -9369.354} C_VEL
LIN {X 0,Y 432.428,Z 152.113,A -85,B 0,C 180,E1 -9372.804,E2 -9372.804} C_VEL
LIN {X 0,Y 432.41,Z 152.114,A -85,B 0,C 180,E1 -9376.479,E2 -9376.479} C_VEL
LIN {X 0,Y 432.336,Z 152.118,A -85,B 0,C 180,E1 -9379.961,E2 -9379.961} C_VEL
LIN {X 0,Y 432.317,Z 152.135,A -85,B 0,C 180,E1 -9382.965,E2 -9382.965} C_VEL
LIN {X 0,Y 432.362,Z 152.115,A -85,B 0,C 180,E1 -9386.033,E2 -9386.033} C_VEL
LIN {X 0,Y 432.341,Z 152.13,A -85,B 0,C 180,E1 -9389.188,E2 -9389.188} C_VEL
LIN {X 0,Y 432.322,Z 152.132,A -85,B 0,C 180,E1 -9392.444,E2 -9392.444} C_VEL
LIN {X 0,Y 432.343,Z 152.124,A -85,B 0,C 180,E1 -9395.632,E2 -9395.632} C_VEL
LIN {X 0,Y 432.337,Z 152.128,A -85,B 0,C 180,E1 -9398.715,E2 -9398.715} C_VEL
LIN {X 0,Y 432.332,Z 152.128,A -85,B 0,C 180,E1 -9401.798,E2 -9401.798} C_VEL
LIN {X 0,Y 432.333,Z 152.129,A -85,B 0,C 180,E1 -9404.348,E2 -9404.348} C_VEL
LIN {X 0,Y 432.32,Z 152.131,A -85,B 0,C 180,E1 -9407.016,E2 -9407.016} C_VEL
LIN {X 0,Y 432.337,Z 152.115,A -85,B 0,C 180,E1 -9409.821,E2 -9409.821} C_VEL
LIN {X 0,Y 432.311,Z 152.131,A -85,B 0,C 180,E1 -9413.023,E2 -9413.023} C_VEL
LIN {X 0,Y 432.36,Z 152.129,A -85,B 0,C 180,E1 -9415.997,E2 -9415.997} C_VEL
LIN {X 0,Y 432.349,Z 152.133,A -85,B 0,C 180,E1 -9419.49,E2 -9419.49} C_VEL
LIN {X 0,Y 432.428,Z 152.284,A -85,B 0,C 180,E1 -9421.359,E2 -9421.359} C_VEL
LIN {X 0,Y 433.967,Z 160.361,A -85,B 0,C 180,E1 -9423.57,E2 -9423.57} C_VEL
LIN {X 0,Y 434.613,Z 165.325,A -85,B 0,C 180,E1 -9424.899,E2 -9424.899} C_VEL
LIN {X 0,Y 433.689,Z 180.791,A -85,B 0,C 180,E1 -9428.616,E2 -9428.616} C_VEL
LIN {X 0,Y 433.064,Z 190.815,A -85,B 0,C 180,E1 -9431.061,E2 -9431.061} C_VEL
LIN {X 0,Y 432.985,Z 192.802,A -85,B 0,C 180,E1 -9431.518,E2 -9431.518} C_VEL
LIN {X 0,Y 433.519,Z 195.913,A -85,B 0,C 180,E1 -9431.647,E2 -9431.647} C_VEL
LIN {X 0,Y 437.261,Z 217.586,A -85,B 0,C 180,E1 -9432.174,E2 -9432.174} C_VEL
LIN {X 0,Y 436.429,Z 297.703,A -85,B 0,C 180,E1 -9433.512,E2 -9433.512} C_VEL
LIN {X 0,Y 436.161,Z 307.598,A -85,B 0,C 180,E1 -9433.772,E2 -9433.772} C_VEL
LIN {X 0,Y 435.783,Z 317.574,A -85,B 0,C 180,E1 -9434.148,E2 -9434.148} C_VEL
LIN {X 0,Y 435.27,Z 327.937,A -85,B 0,C 180,E1 -9434.669,E2 -9434.669} C_VEL
LIN {X 0,Y 434.722,Z 337.07,A -85,B 0,C 180,E1 -9435.249,E2 -9435.249} C_VEL
LIN {X 0,Y 434.192,Z 346.068,A -85,B 0,C 180,E1 -9435.949,E2 -9435.949} C_VEL
LIN {X 0,Y 433.756,Z 353.289,A -85,B 0,C 180,E1 -9436.611,E2 -9436.611} C_VEL
LIN {X 0,Y 433.206,Z 362.195,A -85,B 0,C 180,E1 -9437.587,E2 -9437.587} C_VEL
LIN {X 0,Y 432.738,Z 369.416,A -85,B 0,C 180,E1 -9438.525,E2 -9438.525} C_VEL
LIN {X 0,Y 432.301,Z 375.617,A -85,B 0,C 180,E1 -9439.462,E2 -9439.462} C_VEL
LIN {X 0,Y 431.933,Z 382.155,A -85,B 0,C 180,E1 -9440.636,E2 -9440.636} C_VEL
LIN {X 0,Y 431.681,Z 386.656,A -85,B 0,C 180,E1 -9441.575,E2 -9441.575} C_VEL
LIN {X 0,Y 431.416,Z 392.147,A -85,B 0,C 180,E1 -9442.982,E2 -9442.982} C_VEL
LIN {X 0,Y 431.277,Z 396.469,A -85,B 0,C 180,E1 -9444.389,E2 -9444.389} C_VEL
LIN {X 0,Y 431.271,Z 398.836,A -85,B 0,C 180,E1 -9445.326,E2 -9445.326} C_VEL
LIN {X 0,Y 431.236,Z 402.019,A -85,B 0,C 180,E1 -9447.198,E2 -9447.198} C_VEL
LIN {X 0,Y 431.203,Z 403.074,A -85,B 0,C 180,E1 -9448.132,E2 -9448.132} C_VEL
LIN {X 0,Y 431.17,Z 403.661,A -85,B 0,C 180,E1 -9449.066,E2 -9449.066} C_VEL
LIN {X 0,Y 431.17,Z 403.661,A -85,B 0,C 180,E1 -9450.934,E2 -9450.934} C_VEL
LIN {X 0,Y 431.203,Z 403.074,A -85,B 0,C 180,E1 -9451.868,E2 -9451.868} C_VEL
LIN {X 0,Y 431.187,Z 400.631,A -85,B 0,C 180,E1 -9453.738,E2 -9453.738} C_VEL
LIN {X 0,Y 431.293,Z 397.687,A -85,B 0,C 180,E1 -9455.142,E2 -9455.142} C_VEL
LIN {X 0,Y 431.377,Z 393.7,A -85,B 0,C 180,E1 -9456.548,E2 -9456.548} C_VEL
LIN {X 0,Y 431.565,Z 388.571,A -85,B 0,C 180,E1 -9457.956,E2 -9457.956} C_VEL
LIN {X 0,Y 431.84,Z 383.31,A -85,B 0,C 180,E1 -9459.13,E2 -9459.13} C_VEL
LIN {X 0,Y 432.216,Z 376.993,A -85,B 0,C 180,E1 -9460.303,E2 -9460.303} C_VEL
LIN {X 0,Y 432.598,Z 371.042,A -85,B 0,C 180,E1 -9461.242,E2 -9461.242} C_VEL
LIN {X 0,Y 433.102,Z 364.115,A -85,B 0,C 180,E1 -9462.178,E2 -9462.178} C_VEL
LIN {X 0,Y 433.572,Z 355.933,A -85,B 0,C 180,E1 -9463.116,E2 -9463.116} C_VEL
LIN {X 0,Y 434.115,Z 347.269,A -85,B 0,C 180,E1 -9463.948,E2 -9463.948} C_VEL
LIN {X 0,Y 434.662,Z 338.704,A -85,B 0,C 180,E1 -9464.634,E2 -9464.634} C_VEL
LIN {X 0,Y 435.195,Z 328.944,A -85,B 0,C 180,E1 -9465.274,E2 -9465.274} C_VEL
LIN {X 0,Y 435.679,Z 320.15,A -85,B 0,C 180,E1 -9465.736,E2 -9465.736} C_VEL
LIN {X 0,Y 436.076,Z 310.222,A -85,B 0,C 180,E1 -9466.141,E2 -9466.141} C_VEL
LIN {X 0,Y 436.39,Z 300.367,A -85,B 0,C 180,E1 -9466.43,E2 -9466.43} C_VEL
LIN {X 0,Y 436.806,Z 275.473,A -85,B 0,C 180,E1 -9466.869,E2 -9466.869} C_VEL
LIN {X 0,Y 437.064,Z 215.967,A -85,B 0,C 180,E1 -9467.862,E2 -9467.862} C_VEL
LIN {X 0,Y 433.014,Z 193.14,A -85,B 0,C 180,E1 -9468.445,E2 -9468.445} C_VEL
LIN {X 0,Y 433.008,Z 191.86,A -85,B 0,C 180,E1 -9468.672,E2 -9468.672} C_VEL
LIN {X 0,Y 433.729,Z 179.967,A -85,B 0,C 180,E1 -9471.631,E2 -9471.631} C_VEL
LIN {X 0,Y 434.673,Z 165.539,A -85,B 0,C 180,E1 -9475.117,E2 -9475.117} C_VEL
LIN {X 0,Y 433.63,Z 158.277,A -85,B 0,C 180,E1 -9476.988,E2 -9476.988} C_VEL
LIN {X 0,Y 432.399,Z 152.144,A -85,B 0,C 180,E1 -9478.725,E2 -9478.725} C_VEL
LIN {X 0,Y 432.326,Z 152.128,A -85,B 0,C 180,E1 -9482.293,E2 -9482.293} C_VEL
LIN {X 0,Y 432.341,Z 152.126,A -85,B 0,C 180,E1 -9484.677,E2 -9484.677} C_VEL
LIN {X 0,Y 432.347,Z 152.128,A -85,B 0,C 180,E1 -9488.148,E2 -9488.148} C_VEL
LIN {X 0,Y 432.333,Z 152.122,A -85,B 0,C 180,E1 -9491.601,E2 -9491.601} C_VEL
LIN {X 0,Y 432.334,Z 152.128,A -85,B 0,C 180,E1 -9494.347,E2 -9494.347} C_VEL
LIN {X 0,Y 432.319,Z 152.132,A -85,B 0,C 180,E1 -9497.015,E2 -9497.015} C_VEL
LIN {X 0,Y 432.333,Z 152.124,A -85,B 0,C 180,E1 -9499.82,E2 -9499.82} C_VEL
LIN {X 0,Y 432.305,Z 152.136,A -85,B 0,C 180,E1 -9503.021,E2 -9503.021} C_VEL
LIN {X 0,Y 432.358,Z 152.116,A -85,B 0,C 180,E1 -9505.996,E2 -9505.996} C_VEL
LIN {X 0,Y 432.346,Z 152.13,A -85,B 0,C 180,E1 -9509.489,E2 -9509.489} C_VEL
LIN {X 0,Y 432.389,Z 152.111,A -85,B 0,C 180,E1 -9512.928,E2 -9512.928} C_VEL
LIN {X 0,Y 432.369,Z 152.122,A -85,B 0,C 180,E1 -9516.023,E2 -9516.023} C_VEL
LIN {X 0,Y 432.348,Z 152.122,A -85,B 0,C 180,E1 -9519.045,E2 -9519.045} C_VEL
LIN {X 0,Y 432.375,Z 152.107,A -85,B 0,C 180,E1 -9522.011,E2 -9522.011} C_VEL
LIN {X 0,Y 432.394,Z 152.125,A -85,B 0,C 180,E1 -9524.926,E2 -9524.926} C_VEL
LIN {X 0,Y 432.456,Z 152.108,A -85,B 0,C 180,E1 -9527.803,E2 -9527.803} C_VEL
LIN {X 0,Y 432.489,Z 152.096,A -85,B 0,C 180,E1 -9531.59,E2 -9531.59} C_VEL
LIN {X 0,Y 432.594,Z 152.099,A -85,B 0,C 180,E1 -9534.406,E2 -9534.406} C_VEL
LIN {X 0,Y 432.6,Z 152.091,A -85,B 0,C 180,E1 -9538.138,E2 -9538.138} C_VEL
LIN {X 0,Y 432.728,Z 152.062,A -85,B 0,C 180,E1 -9539.999,E2 -9539.999} C_VEL
LIN {X 0,Y 432.601,Z 152.094,A -85,B 0,C 180,E1 -9542.793,E2 -9542.793} C_VEL
LIN {X 0,Y 432.569,Z 152.098,A -85,B 0,C 180,E1 -9546.53,E2 -9546.53} C_VEL
LIN {X 0,Y 432.438,Z 152.099,A -85,B 0,C 180,E1 -9549.353,E2 -9549.353} C_VEL
LIN {X 0,Y 432.426,Z 152.115,A -85,B 0,C 180,E1 -9552.803,E2 -9552.803} C_VEL
LIN {X 0,Y 432.408,Z 152.115,A -85,B 0,C 180,E1 -9556.479,E2 -9556.479} C_VEL
LIN {X 0,Y 432.334,Z 152.117,A -85,B 0,C 180,E1 -9559.96,E2 -9559.96} C_VEL
LIN {X 0,Y 432.315,Z 152.131,A -85,B 0,C 180,E1 -9562.964,E2 -9562.964} C_VEL
LIN {X 0,Y 432.36,Z 152.117,A -85,B 0,C 180,E1 -9566.032,E2 -9566.032} C_VEL
LIN {X 0,Y 432.343,Z 152.123,A -85,B 0,C 180,E1 -9569.187,E2 -9569.187} C_VEL
LIN {X 0,Y 432.32,Z 152.129,A -85,B 0,C 180,E1 -9572.293,E2 -9572.293} C_VEL
LIN {X 0,Y 432.336,Z 152.115,A -85,B 0,C 180,E1 -9574.677,E2 -9574.677} C_VEL
LIN {X 0,Y 432.342,Z 152.128,A -85,B 0,C 180,E1 -9578.149,E2 -9578.149} C_VEL
LIN {X 0,Y 432.329,Z 152.13,A -85,B 0,C 180,E1 -9581.602,E2 -9581.602} C_VEL
LIN {X 0,Y 432.336,Z 152.128,A -85,B 0,C 180,E1 -9584.346,E2 -9584.346} C_VEL
LIN {X 0,Y 432.319,Z 152.108,A -85,B 0,C 180,E1 -9587.015,E2 -9587.015} C_VEL
LIN {X 0,Y 432.328,Z 152.124,A -85,B 0,C 180,E1 -9589.821,E2 -9589.821} C_VEL
LIN {X 0,Y 432.311,Z 152.133,A -85,B 0,C 180,E1 -9593.023,E2 -9593.023} C_VEL
LIN {X 0,Y 432.355,Z 152.114,A -85,B 0,C 180,E1 -9595.996,E2 -9595.996} C_VEL
LIN {X 0,Y 432.392,Z 152.117,A -85,B 0,C 180,E1 -9599.744,E2 -9599.744} C_VEL
LIN {X 0,Y 432.395,Z 152.124,A -85,B 0,C 180,E1 -9603.372,E2 -9603.372} C_VEL
LIN {X 0,Y 432.368,Z 152.127,A -85,B 0,C 180,E1 -9606.023,E2 -9606.023} C_VEL
LIN {X 0,Y 432.346,Z 152.132,A -85,B 0,C 180,E1 -9609.046,E2 -9609.046} C_VEL
LIN {X 0,Y 432.374,Z 152.129,A -85,B 0,C 180,E1 -9612.011,E2 -9612.011} C_VEL
LIN {X 0,Y 432.392,Z 152.126,A -85,B 0,C 180,E1 -9614.927,E2 -9614.927} C_VEL
LIN {X 0,Y 432.456,Z 152.119,A -85,B 0,C 180,E1 -9617.803,E2 -9617.803} C_VEL
LIN {X 0,Y 432.488,Z 152.115,A -85,B 0,C 180,E1 -9621.59,E2 -9621.59} C_VEL
LIN {X 0,Y 432.595,Z 152.102,A -85,B 0,C 180,E1 -9624.406,E2 -9624.406} C_VEL
LIN {X 0,Y 432.603,Z 152.101,A -85,B 0,C 180,E1 -9628.138,E2 -9628.138} C_VEL
LIN {X 0,Y 432.731,Z 152.086,A -85,B 0,C 180,E1 -9630,E2 -9630} C_VEL
LIN {X 0,Y 432.602,Z 152.099,A -85,B 0,C 180,E1 -9632.794,E2 -9632.794} C_VEL
LIN {X 0,Y 432.46,Z 152.117,A -85,B 0,C 180,E1 -9635.02,E2 -9635.02} C_VEL
LIN {X 0,Y 431.9,Z 152.189,A -85,B 0,C 180,E1 -9635.799,E2 -9635.799} C_VEL
LIN {X 0,Y 429.055,Z 152.542,A -85,B 0,C 180,E1 -9637.064,E2 -9637.064} C_VEL
LIN {X 0,Y 426.572,Z 152.852,A -85,B 0,C 180,E1 -9638.085,E2 -9638.085} C_VEL
LIN {X 0,Y 425.491,Z 152.986,A -85,B 0,C 180,E1 -9638.875,E2 -9638.875} C_VEL
LIN {X 0,Y 425.4,Z 152.997,A -85,B 0,C 180,E1 -9639.143,E2 -9639.143} C_VEL
LIN {X 0,Y 425.39,Z 152.998,A -85,B 0,C 180,E1 -9642.904,E2 -9642.904} C_VEL
LIN {X 0,Y 425.358,Z 153.001,A -85,B 0,C 180,E1 -9646.605,E2 -9646.605} C_VEL
LIN {X 0,Y 425.325,Z 153.008,A -85,B 0,C 180,E1 -9649.636,E2 -9649.636} C_VEL
LIN {X 0,Y 425.303,Z 153.011,A -85,B 0,C 180,E1 -9653.365,E2 -9653.365} C_VEL
LIN {X 0,Y 425.344,Z 153.004,A -85,B 0,C 180,E1 -9656.844,E2 -9656.844} C_VEL
LIN {X 0,Y 425.315,Z 152.995,A -85,B 0,C 180,E1 -9659.717,E2 -9659.717} C_VEL
LIN {X 0,Y 425.28,Z 153.003,A -85,B 0,C 180,E1 -9663.048,E2 -9663.048} C_VEL
LIN {X 0,Y 425.279,Z 153.001,A -85,B 0,C 180,E1 -9665.929,E2 -9665.929} C_VEL
LIN {X 0,Y 425.291,Z 153.006,A -85,B 0,C 180,E1 -9669.043,E2 -9669.043} C_VEL
LIN {X 0,Y 425.272,Z 152.98,A -85,B 0,C 180,E1 -9672.653,E2 -9672.653} C_VEL
LIN {X 0,Y 425.263,Z 153.009,A -85,B 0,C 180,E1 -9676.045,E2 -9676.045} C_VEL
LIN {X 0,Y 425.271,Z 153.005,A -85,B 0,C 180,E1 -9678.622,E2 -9678.622} C_VEL
LIN {X 0,Y 425.308,Z 153.007,A -85,B 0,C 180,E1 -9681.103,E2 -9681.103} C_VEL
LIN {X 0,Y 425.295,Z 152.998,A -85,B 0,C 180,E1 -9684.664,E2 -9684.664} C_VEL
LIN {X 0,Y 425.261,Z 153.011,A -85,B 0,C 180,E1 -9688.073,E2 -9688.073} C_VEL
LIN {X 0,Y 425.33,Z 152.994,A -85,B 0,C 180,E1 -9691.368,E2 -9691.368} C_VEL
LIN {X 0,Y 425.292,Z 153.006,A -85,B 0,C 180,E1 -9694.555,E2 -9694.555} C_VEL
LIN {X 0,Y 425.283,Z 153.008,A -85,B 0,C 180,E1 -9697.662,E2 -9697.662} C_VEL
LIN {X 0,Y 425.357,Z 152.979,A -85,B 0,C 180,E1 -9700.704,E2 -9700.704} C_VEL
LIN {X 0,Y 425.384,Z 152.992,A -85,B 0,C 180,E1 -9703.689,E2 -9703.689} C_VEL
LIN {X 0,Y 425.408,Z 152.992,A -85,B 0,C 180,E1 -9707.599,E2 -9707.599} C_VEL
LIN {X 0,Y 425.438,Z 152.973,A -85,B 0,C 180,E1 -9711.45,E2 -9711.45} C_VEL
LIN {X 0,Y 425.55,Z 152.975,A -85,B 0,C 180,E1 -9714.314,E2 -9714.314} C_VEL
LIN {X 0,Y 425.572,Z 152.959,A -85,B 0,C 180,E1 -9718.108,E2 -9718.108} C_VEL
LIN {X 0,Y 425.698,Z 152.937,A -85,B 0,C 180,E1 -9720.001,E2 -9720.001} C_VEL
LIN {X 0,Y 425.543,Z 152.97,A -85,B 0,C 180,E1 -9722.84,E2 -9722.84} C_VEL
LIN {X 0,Y 425.528,Z 152.974,A -85,B 0,C 180,E1 -9726.639,E2 -9726.639} C_VEL
LIN {X 0,Y 425.397,Z 152.974,A -85,B 0,C 180,E1 -9729.51,E2 -9729.51} C_VEL
LIN {X 0,Y 425.391,Z 152.991,A -85,B 0,C 180,E1 -9732.904,E2 -9732.904} C_VEL
LIN {X 0,Y 425.359,Z 152.993,A -85,B 0,C 180,E1 -9736.606,E2 -9736.606} C_VEL
LIN {X 0,Y 425.326,Z 152.991,A -85,B 0,C 180,E1 -9739.636,E2 -9739.636} C_VEL
LIN {X 0,Y 425.305,Z 153.005,A -85,B 0,C 180,E1 -9743.366,E2 -9743.366} C_VEL
LIN {X 0,Y 425.345,Z 152.987,A -85,B 0,C 180,E1 -9746.845,E2 -9746.845} C_VEL
LIN {X 0,Y 425.289,Z 153.005,A -85,B 0,C 180,E1 -9749.72,E2 -9749.72} C_VEL
LIN {X 0,Y 425.281,Z 153,A -85,B 0,C 180,E1 -9753.049,E2 -9753.049} C_VEL
LIN {X 0,Y 425.281,Z 153.004,A -85,B 0,C 180,E1 -9755.929,E2 -9755.929} C_VEL
LIN {X 0,Y 425.28,Z 153.003,A -85,B 0,C 180,E1 -9759.041,E2 -9759.041} C_VEL
LIN {X 0,Y 425.289,Z 153.006,A -85,B 0,C 180,E1 -9761.959,E2 -9761.959} C_VEL
LIN {X 0,Y 425.285,Z 153.006,A -85,B 0,C 180,E1 -9765.284,E2 -9765.284} C_VEL
LIN {X 0,Y 425.275,Z 152.999,A -85,B 0,C 180,E1 -9768.622,E2 -9768.622} C_VEL
LIN {X 0,Y 425.314,Z 153.002,A -85,B 0,C 180,E1 -9771.104,E2 -9771.104} C_VEL
LIN {X 0,Y 425.3,Z 152.998,A -85,B 0,C 180,E1 -9774.665,E2 -9774.665} C_VEL
LIN {X 0,Y 425.266,Z 153.007,A -85,B 0,C 180,E1 -9778.074,E2 -9778.074} C_VEL
LIN {X 0,Y 425.376,Z 153.202,A -85,B 0,C 180,E1 -9781.124,E2 -9781.124} C_VEL
LIN {X 0,Y 427.066,Z 162.114,A -85,B 0,C 180,E1 -9783.62,E2 -9783.62} C_VEL
LIN {X 0,Y 427.62,Z 167.162,A -85,B 0,C 180,E1 -9784.963,E2 -9784.963} C_VEL
LIN {X 0,Y 426.698,Z 181.66,A -85,B 0,C 180,E1 -9788.502,E2 -9788.502} C_VEL
LIN {X 0,Y 426.024,Z 192.611,A -85,B 0,C 180,E1 -9791.205,E2 -9791.205} C_VEL
LIN {X 0,Y 426.467,Z 195.448,A -85,B 0,C 180,E1 -9791.327,E2 -9791.327} C_VEL
LIN {X 0,Y 430.501,Z 218.198,A -85,B 0,C 180,E1 -9791.898,E2 -9791.898} C_VEL
LIN {X 0,Y 429.637,Z 297.512,A -85,B 0,C 180,E1 -9793.243,E2 -9793.243} C_VEL
LIN {X 0,Y 429.348,Z 307.407,A -85,B 0,C 180,E1 -9793.507,E2 -9793.507} C_VEL
LIN {X 0,Y 428.942,Z 317.382,A -85,B 0,C 180,E1 -9793.888,E2 -9793.888} C_VEL
LIN {X 0,Y 428.415,Z 327.745,A -85,B 0,C 180,E1 -9794.418,E2 -9794.418} C_VEL
LIN {X 0,Y 427.835,Z 336.878,A -85,B 0,C 180,E1 -9795.006,E2 -9795.006} C_VEL
LIN {X 0,Y 427.274,Z 345.876,A -85,B 0,C 180,E1 -9795.716,E2 -9795.716} C_VEL
LIN {X 0,Y 426.779,Z 353.884,A -85,B 0,C 180,E1 -9796.473,E2 -9796.473} C_VEL
LIN {X 0,Y 426.247,Z 362.003,A -85,B 0,C 180,E1 -9797.381,E2 -9797.381} C_VEL
LIN {X 0,Y 425.764,Z 369.224,A -85,B 0,C 180,E1 -9798.334,E2 -9798.334} C_VEL
LIN {X 0,Y 425.286,Z 375.424,A -85,B 0,C 180,E1 -9799.286,E2 -9799.286} C_VEL
LIN {X 0,Y 424.874,Z 381.962,A -85,B 0,C 180,E1 -9800.479,E2 -9800.479} C_VEL
LIN {X 0,Y 424.635,Z 386.464,A -85,B 0,C 180,E1 -9801.434,E2 -9801.434} C_VEL
LIN {X 0,Y 424.34,Z 391.954,A -85,B 0,C 180,E1 -9802.865,E2 -9802.865} C_VEL
LIN {X 0,Y 424.189,Z 396.277,A -85,B 0,C 180,E1 -9804.295,E2 -9804.295} C_VEL
LIN {X 0,Y 424.2,Z 398.644,A -85,B 0,C 180,E1 -9805.248,E2 -9805.248} C_VEL
LIN {X 0,Y 424.132,Z 401.827,A -85,B 0,C 180,E1 -9807.151,E2 -9807.151} C_VEL
LIN {X 0,Y 424.129,Z 402.883,A -85,B 0,C 180,E1 -9808.101,E2 -9808.101} C_VEL
LIN {X 0,Y 424.09,Z 403.47,A -85,B 0,C 180,E1 -9809.05,E2 -9809.05} C_VEL
LIN {X 0,Y 424.09,Z 403.47,A -85,B 0,C 180,E1 -9810.95,E2 -9810.95} C_VEL
LIN {X 0,Y 424.129,Z 402.883,A -85,B 0,C 180,E1 -9811.899,E2 -9811.899} C_VEL
LIN {X 0,Y 424.099,Z 400.44,A -85,B 0,C 180,E1 -9813.801,E2 -9813.801} C_VEL
LIN {X 0,Y 424.205,Z 397.495,A -85,B 0,C 180,E1 -9815.228,E2 -9815.228} C_VEL
LIN {X 0,Y 424.3,Z 393.508,A -85,B 0,C 180,E1 -9816.658,E2 -9816.658} C_VEL
LIN {X 0,Y 424.516,Z 388.379,A -85,B 0,C 180,E1 -9818.089,E2 -9818.089} C_VEL
LIN {X 0,Y 424.806,Z 383.118,A -85,B 0,C 180,E1 -9819.283,E2 -9819.283} C_VEL
LIN {X 0,Y 425.183,Z 376.8,A -85,B 0,C 180,E1 -9820.476,E2 -9820.476} C_VEL
LIN {X 0,Y 425.628,Z 370.85,A -85,B 0,C 180,E1 -9821.428,E2 -9821.428} C_VEL
LIN {X 0,Y 426.132,Z 363.923,A -85,B 0,C 180,E1 -9822.38,E2 -9822.38} C_VEL
LIN {X 0,Y 426.628,Z 355.741,A -85,B 0,C 180,E1 -9823.334,E2 -9823.334} C_VEL
LIN {X 0,Y 427.211,Z 346.97,A -85,B 0,C 180,E1 -9824.188,E2 -9824.188} C_VEL
LIN {X 0,Y 427.79,Z 338.512,A -85,B 0,C 180,E1 -9824.874,E2 -9824.874} C_VEL
LIN {X 0,Y 428.283,Z 329.759,A -85,B 0,C 180,E1 -9825.465,E2 -9825.465} C_VEL
LIN {X 0,Y 428.857,Z 319.959,A -85,B 0,C 180,E1 -9825.993,E2 -9825.993} C_VEL
LIN {X 0,Y 429.277,Z 310.03,A -85,B 0,C 180,E1 -9826.404,E2 -9826.404} C_VEL
LIN {X 0,Y 429.593,Z 300.176,A -85,B 0,C 180,E1 -9826.697,E2 -9826.697} C_VEL
LIN {X 0,Y 429.991,Z 275.378,A -85,B 0,C 180,E1 -9827.143,E2 -9827.143} C_VEL
LIN {X 0,Y 430.367,Z 217.243,A -85,B 0,C 180,E1 -9828.124,E2 -9828.124} C_VEL
LIN {X 0,Y 426.04,Z 192.879,A -85,B 0,C 180,E1 -9828.763,E2 -9828.763} C_VEL
LIN {X 0,Y 426.052,Z 191.578,A -85,B 0,C 180,E1 -9829.013,E2 -9829.013} C_VEL
LIN {X 0,Y 426.804,Z 179.792,A -85,B 0,C 180,E1 -9832,E2 -9832} C_VEL
LIN {X 0,Y 427.716,Z 166.467,A -85,B 0,C 180,E1 -9835.291,E2 -9835.291} C_VEL
LIN {X 0,Y 426.602,Z 159.26,A -85,B 0,C 180,E1 -9837.174,E2 -9837.174} C_VEL
LIN {X 0,Y 425.33,Z 153.02,A -85,B 0,C 180,E1 -9838.982,E2 -9838.982} C_VEL
LIN {X 0,Y 425.283,Z 153.006,A -85,B 0,C 180,E1 -9842.562,E2 -9842.562} C_VEL
LIN {X 0,Y 425.3,Z 152.999,A -85,B 0,C 180,E1 -9845.335,E2 -9845.335} C_VEL
LIN {X 0,Y 425.301,Z 153.002,A -85,B 0,C 180,E1 -9849.043,E2 -9849.043} C_VEL
LIN {X 0,Y 425.275,Z 153.008,A -85,B 0,C 180,E1 -9852.652,E2 -9852.652} C_VEL
LIN {X 0,Y 425.261,Z 153.011,A -85,B 0,C 180,E1 -9856.043,E2 -9856.043} C_VEL
LIN {X 0,Y 425.273,Z 153.008,A -85,B 0,C 180,E1 -9858.621,E2 -9858.621} C_VEL
LIN {X 0,Y 425.296,Z 153.002,A -85,B 0,C 180,E1 -9861.101,E2 -9861.101} C_VEL
LIN {X 0,Y 425.298,Z 153.002,A -85,B 0,C 180,E1 -9864.663,E2 -9864.663} C_VEL
LIN {X 0,Y 425.263,Z 153.008,A -85,B 0,C 180,E1 -9868.072,E2 -9868.072} C_VEL
LIN {X 0,Y 425.33,Z 152.995,A -85,B 0,C 180,E1 -9871.367,E2 -9871.367} C_VEL
LIN {X 0,Y 425.293,Z 152.997,A -85,B 0,C 180,E1 -9874.554,E2 -9874.554} C_VEL
LIN {X 0,Y 425.286,Z 153.005,A -85,B 0,C 180,E1 -9877.661,E2 -9877.661} C_VEL
LIN {X 0,Y 425.36,Z 152.983,A -85,B 0,C 180,E1 -9880.703,E2 -9880.703} C_VEL
LIN {X 0,Y 425.386,Z 152.989,A -85,B 0,C 180,E1 -9883.688,E2 -9883.688} C_VEL
LIN {X 0,Y 425.409,Z 152.985,A -85,B 0,C 180,E1 -9887.598,E2 -9887.598} C_VEL
LIN {X 0,Y 425.439,Z 152.974,A -85,B 0,C 180,E1 -9891.449,E2 -9891.449} C_VEL
LIN {X 0,Y 425.551,Z 152.975,A -85,B 0,C 180,E1 -9894.313,E2 -9894.313} C_VEL
LIN {X 0,Y 425.569,Z 152.967,A -85,B 0,C 180,E1 -9898.107,E2 -9898.107} C_VEL
LIN {X 0,Y 425.698,Z 152.937,A -85,B 0,C 180,E1 -9899.999,E2 -9899.999} C_VEL
LIN {X 0,Y 425.553,Z 152.971,A -85,B 0,C 180,E1 -9902.839,E2 -9902.839} C_VEL
LIN {X 0,Y 425.527,Z 152.974,A -85,B 0,C 180,E1 -9906.638,E2 -9906.638} C_VEL
LIN {X 0,Y 425.397,Z 152.976,A -85,B 0,C 180,E1 -9909.509,E2 -9909.509} C_VEL
LIN {X 0,Y 425.389,Z 152.991,A -85,B 0,C 180,E1 -9912.903,E2 -9912.903} C_VEL
LIN {X 0,Y 425.357,Z 152.993,A -85,B 0,C 180,E1 -9916.605,E2 -9916.605} C_VEL
LIN {X 0,Y 425.324,Z 152.986,A -85,B 0,C 180,E1 -9919.635,E2 -9919.635} C_VEL
LIN {X 0,Y 425.303,Z 153.007,A -85,B 0,C 180,E1 -9923.365,E2 -9923.365} C_VEL
LIN {X 0,Y 425.344,Z 152.987,A -85,B 0,C 180,E1 -9926.844,E2 -9926.844} C_VEL
LIN {X 0,Y 425.31,Z 153.006,A -85,B 0,C 180,E1 -9929.717,E2 -9929.717} C_VEL
LIN {X 0,Y 425.277,Z 153.008,A -85,B 0,C 180,E1 -9933.048,E2 -9933.048} C_VEL
LIN {X 0,Y 425.279,Z 153.008,A -85,B 0,C 180,E1 -9935.929,E2 -9935.929} C_VEL
LIN {X 0,Y 425.296,Z 153.009,A -85,B 0,C 180,E1 -9939.044,E2 -9939.044} C_VEL
LIN {X 0,Y 425.273,Z 153.008,A -85,B 0,C 180,E1 -9942.652,E2 -9942.652} C_VEL
LIN {X 0,Y 425.263,Z 152.997,A -85,B 0,C 180,E1 -9946.045,E2 -9946.045} C_VEL
LIN {X 0,Y 425.268,Z 152.981,A -85,B 0,C 180,E1 -9948.621,E2 -9948.621} C_VEL
LIN {X 0,Y 425.304,Z 153.007,A -85,B 0,C 180,E1 -9951.102,E2 -9951.102} C_VEL
LIN {X 0,Y 425.296,Z 152.993,A -85,B 0,C 180,E1 -9954.664,E2 -9954.664} C_VEL
LIN {X 0,Y 425.27,Z 153.01,A -85,B 0,C 180,E1 -9958.074,E2 -9958.074} C_VEL
LIN {X 0,Y 425.334,Z 152.995,A -85,B 0,C 180,E1 -9961.368,E2 -9961.368} C_VEL
LIN {X 0,Y 425.292,Z 153.012,A -85,B 0,C 180,E1 -9964.555,E2 -9964.555} C_VEL
LIN {X 0,Y 425.284,Z 153.01,A -85,B 0,C 180,E1 -9967.661,E2 -9967.661} C_VEL
LIN {X 0,Y 425.358,Z 153.004,A -85,B 0,C 180,E1 -9970.704,E2 -9970.704} C_VEL
LIN {X 0,Y 425.385,Z 152.998,A -85,B 0,C 180,E1 -9973.688,E2 -9973.688} C_VEL
LIN {X 0,Y 425.408,Z 152.996,A -85,B 0,C 180,E1 -9977.598,E2 -9977.598} C_VEL
LIN {X 0,Y 425.439,Z 152.993,A -85,B 0,C 180,E1 -9981.45,E2 -9981.45} C_VEL
LIN {X 0,Y 425.551,Z 152.979,A -85,B 0,C 180,E1 -9984.313,E2 -9984.313} C_VEL
LIN {X 0,Y 425.572,Z 152.976,A -85,B 0,C 180,E1 -9988.107,E2 -9988.107} C_VEL
LIN {X 0,Y 425.7,Z 152.961,A -85,B 0,C 180,E1 -9990,E2 -9990} C_VEL
LIN {X 0,Y 425.554,Z 152.977,A -85,B 0,C 180,E1 -9992.84,E2 -9992.84} C_VEL
LIN {X 0,Y 425.528,Z 152.981,A -85,B 0,C 180,E1 -9996.639,E2 -9996.639} C_VEL
LIN {X 0,Y 425.4,Z 152.997,A -85,B 0,C 180,E1 -9999.143,E2 -9999.143} C_VEL
LIN {X 0,Y 424.727,Z 153.082,A -85,B 0,C 180,E1 -9999.933,E2 -9999.933} C_VEL
LIN {X 0,Y 421.88,Z 153.436,A -85,B 0,C 180,E1 -10001.216,E2 -10001.216} C_VEL
LIN {X 0,Y 419.464,Z 153.737,A -85,B 0,C 180,E1 -10002.252,E2 -10002.252} C_VEL
LIN {X 0,Y 418.413,Z 153.867,A -85,B 0,C 180,E1 -10003.053,E2 -10003.053} C_VEL
LIN {X 0,Y 418.319,Z 153.879,A -85,B 0,C 180,E1 -10003.324,E2 -10003.324} C_VEL
LIN {X 0,Y 418.309,Z 153.879,A -85,B 0,C 180,E1 -10006.736,E2 -10006.736} C_VEL
LIN {X 0,Y 418.267,Z 153.887,A -85,B 0,C 180,E1 -10009.79,E2 -10009.79} C_VEL
LIN {X 0,Y 418.234,Z 153.889,A -85,B 0,C 180,E1 -10012.736,E2 -10012.736} C_VEL
LIN {X 0,Y 418.267,Z 153.885,A -85,B 0,C 180,E1 -10015.904,E2 -10015.904} C_VEL
LIN {X 0,Y 418.271,Z 153.871,A -85,B 0,C 180,E1 -10019.161,E2 -10019.161} C_VEL
LIN {X 0,Y 418.256,Z 153.881,A -85,B 0,C 180,E1 -10022.845,E2 -10022.845} C_VEL
LIN {X 0,Y 418.243,Z 153.878,A -85,B 0,C 180,E1 -10026.239,E2 -10026.239} C_VEL
LIN {X 0,Y 418.244,Z 153.878,A -85,B 0,C 180,E1 -10029.682,E2 -10029.682} C_VEL
LIN {X 0,Y 418.226,Z 153.855,A -85,B 0,C 180,E1 -10032.321,E2 -10032.321} C_VEL
LIN {X 0,Y 418.237,Z 153.885,A -85,B 0,C 180,E1 -10035.11,E2 -10035.11} C_VEL
LIN {X 0,Y 418.237,Z 153.883,A -85,B 0,C 180,E1 -10037.767,E2 -10037.767} C_VEL
LIN {X 0,Y 418.252,Z 153.881,A -85,B 0,C 180,E1 -10040.619,E2 -10040.619} C_VEL
LIN {X 0,Y 418.241,Z 153.884,A -85,B 0,C 180,E1 -10043.976,E2 -10043.976} C_VEL
LIN {X 0,Y 418.253,Z 153.882,A -85,B 0,C 180,E1 -10047.156,E2 -10047.156} C_VEL
LIN {X 0,Y 418.266,Z 153.876,A -85,B 0,C 180,E1 -10050.839,E2 -10050.839} C_VEL
LIN {X 0,Y 418.267,Z 153.873,A -85,B 0,C 180,E1 -10054.096,E2 -10054.096} C_VEL
LIN {X 0,Y 418.234,Z 153.885,A -85,B 0,C 180,E1 -10057.264,E2 -10057.264} C_VEL
LIN {X 0,Y 418.278,Z 153.863,A -85,B 0,C 180,E1 -10060.365,E2 -10060.365} C_VEL
LIN {X 0,Y 418.313,Z 153.87,A -85,B 0,C 180,E1 -10063.405,E2 -10063.405} C_VEL
LIN {X 0,Y 418.342,Z 153.869,A -85,B 0,C 180,E1 -10067,E2 -10067} C_VEL
LIN {X 0,Y 418.337,Z 153.854,A -85,B 0,C 180,E1 -10070.329,E2 -10070.329} C_VEL
LIN {X 0,Y 418.509,Z 153.848,A -85,B 0,C 180,E1 -10072.28,E2 -10072.28} C_VEL
LIN {X 0,Y 418.509,Z 153.853,A -85,B 0,C 180,E1 -10074.218,E2 -10074.218} C_VEL
LIN {X 0,Y 418.541,Z 153.835,A -85,B 0,C 180,E1 -10078.076,E2 -10078.076} C_VEL
LIN {X 0,Y 418.667,Z 153.812,A -85,B 0,C 180,E1 -10080.001,E2 -10080.001} C_VEL
LIN {X 0,Y 418.498,Z 153.848,A -85,B 0,C 180,E1 -10082.888,E2 -10082.888} C_VEL
LIN {X 0,Y 418.491,Z 153.851,A -85,B 0,C 180,E1 -10086.752,E2 -10086.752} C_VEL
LIN {X 0,Y 418.338,Z 153.853,A -85,B 0,C 180,E1 -10089.672,E2 -10089.672} C_VEL
LIN {X 0,Y 418.344,Z 153.869,A -85,B 0,C 180,E1 -10093.001,E2 -10093.001} C_VEL
LIN {X 0,Y 418.311,Z 153.872,A -85,B 0,C 180,E1 -10096.736,E2 -10096.736} C_VEL
LIN {X 0,Y 418.268,Z 153.87,A -85,B 0,C 180,E1 -10099.791,E2 -10099.791} C_VEL
LIN {X 0,Y 418.236,Z 153.886,A -85,B 0,C 180,E1 -10102.737,E2 -10102.737} C_VEL
LIN {X 0,Y 418.269,Z 153.87,A -85,B 0,C 180,E1 -10105.905,E2 -10105.905} C_VEL
LIN {X 0,Y 418.263,Z 153.884,A -85,B 0,C 180,E1 -10109.163,E2 -10109.163} C_VEL
LIN {X 0,Y 418.256,Z 153.877,A -85,B 0,C 180,E1 -10112.845,E2 -10112.845} C_VEL
LIN {X 0,Y 418.244,Z 153.882,A -85,B 0,C 180,E1 -10116.238,E2 -10116.238} C_VEL
LIN {X 0,Y 418.244,Z 153.877,A -85,B 0,C 180,E1 -10119.683,E2 -10119.683} C_VEL
LIN {X 0,Y 418.229,Z 153.889,A -85,B 0,C 180,E1 -10122.322,E2 -10122.322} C_VEL
LIN {X 0,Y 418.236,Z 153.884,A -85,B 0,C 180,E1 -10125.109,E2 -10125.109} C_VEL
LIN {X 0,Y 418.24,Z 153.886,A -85,B 0,C 180,E1 -10127.767,E2 -10127.767} C_VEL
LIN {X 0,Y 418.258,Z 153.873,A -85,B 0,C 180,E1 -10130.619,E2 -10130.619} C_VEL
LIN {X 0,Y 418.245,Z 153.879,A -85,B 0,C 180,E1 -10133.976,E2 -10133.976} C_VEL
LIN {X 0,Y 418.259,Z 153.882,A -85,B 0,C 180,E1 -10137.157,E2 -10137.157} C_VEL
LIN {X 0,Y 418.306,Z 154.026,A -85,B 0,C 180,E1 -10140.842,E2 -10140.842} C_VEL
LIN {X 0,Y 419.902,Z 161.975,A -85,B 0,C 180,E1 -10143.134,E2 -10143.134} C_VEL
LIN {X 0,Y 420.657,Z 168.463,A -85,B 0,C 180,E1 -10144.894,E2 -10144.894} C_VEL
LIN {X 0,Y 419.716,Z 182.529,A -85,B 0,C 180,E1 -10148.384,E2 -10148.384} C_VEL
LIN {X 0,Y 419.051,Z 192.419,A -85,B 0,C 180,E1 -10150.88,E2 -10150.88} C_VEL
LIN {X 0,Y 419.608,Z 195.7,A -85,B 0,C 180,E1 -10151.019,E2 -10151.019} C_VEL
LIN {X 0,Y 423.66,Z 218.275,A -85,B 0,C 180,E1 -10151.6,E2 -10151.6} C_VEL
LIN {X 0,Y 422.862,Z 297.321,A -85,B 0,C 180,E1 -10152.967,E2 -10152.967} C_VEL
LIN {X 0,Y 422.547,Z 307.215,A -85,B 0,C 180,E1 -10153.234,E2 -10153.234} C_VEL
LIN {X 0,Y 422.103,Z 317.19,A -85,B 0,C 180,E1 -10153.62,E2 -10153.62} C_VEL
LIN {X 0,Y 421.581,Z 327.553,A -85,B 0,C 180,E1 -10154.158,E2 -10154.158} C_VEL
LIN {X 0,Y 420.971,Z 336.686,A -85,B 0,C 180,E1 -10154.755,E2 -10154.755} C_VEL
LIN {X 0,Y 420.394,Z 345.684,A -85,B 0,C 180,E1 -10155.477,E2 -10155.477} C_VEL
LIN {X 0,Y 419.853,Z 353.482,A -85,B 0,C 180,E1 -10156.222,E2 -10156.222} C_VEL
LIN {X 0,Y 419.283,Z 361.81,A -85,B 0,C 180,E1 -10157.168,E2 -10157.168} C_VEL
LIN {X 0,Y 418.784,Z 369.031,A -85,B 0,C 180,E1 -10158.137,E2 -10158.137} C_VEL
LIN {X 0,Y 418.291,Z 375.232,A -85,B 0,C 180,E1 -10159.105,E2 -10159.105} C_VEL
LIN {X 0,Y 417.831,Z 381.769,A -85,B 0,C 180,E1 -10160.317,E2 -10160.317} C_VEL
LIN {X 0,Y 417.571,Z 386.271,A -85,B 0,C 180,E1 -10161.288,E2 -10161.288} C_VEL
LIN {X 0,Y 417.266,Z 391.762,A -85,B 0,C 180,E1 -10162.743,E2 -10162.743} C_VEL
LIN {X 0,Y 417.107,Z 396.085,A -85,B 0,C 180,E1 -10164.198,E2 -10164.198} C_VEL
LIN {X 0,Y 417.107,Z 398.452,A -85,B 0,C 180,E1 -10165.167,E2 -10165.167} C_VEL
LIN {X 0,Y 417.028,Z 401.635,A -85,B 0,C 180,E1 -10167.102,E2 -10167.102} C_VEL
LIN {X 0,Y 417.057,Z 402.692,A -85,B 0,C 180,E1 -10168.069,E2 -10168.069} C_VEL
LIN {X 0,Y 417.012,Z 403.279,A -85,B 0,C 180,E1 -10169.034,E2 -10169.034} C_VEL
LIN {X 0,Y 417.012,Z 403.279,A -85,B 0,C 180,E1 -10170.966,E2 -10170.966} C_VEL
LIN {X 0,Y 417.057,Z 402.692,A -85,B 0,C 180,E1 -10171.931,E2 -10171.931} C_VEL
LIN {X 0,Y 417.014,Z 400.248,A -85,B 0,C 180,E1 -10173.865,E2 -10173.865} C_VEL
LIN {X 0,Y 417.12,Z 397.303,A -85,B 0,C 180,E1 -10175.317,E2 -10175.317} C_VEL
LIN {X 0,Y 417.232,Z 393.316,A -85,B 0,C 180,E1 -10176.771,E2 -10176.771} C_VEL
LIN {X 0,Y 417.458,Z 388.187,A -85,B 0,C 180,E1 -10178.227,E2 -10178.227} C_VEL
LIN {X 0,Y 417.77,Z 382.925,A -85,B 0,C 180,E1 -10179.44,E2 -10179.44} C_VEL
LIN {X 0,Y 418.159,Z 376.607,A -85,B 0,C 180,E1 -10180.654,E2 -10180.654} C_VEL
LIN {X 0,Y 418.634,Z 370.657,A -85,B 0,C 180,E1 -10181.622,E2 -10181.622} C_VEL
LIN {X 0,Y 419.168,Z 363.73,A -85,B 0,C 180,E1 -10182.589,E2 -10182.589} C_VEL
LIN {X 0,Y 419.708,Z 355.549,A -85,B 0,C 180,E1 -10183.558,E2 -10183.558} C_VEL
LIN {X 0,Y 420.295,Z 346.9,A -85,B 0,C 180,E1 -10184.415,E2 -10184.415} C_VEL
LIN {X 0,Y 420.905,Z 338.319,A -85,B 0,C 180,E1 -10185.123,E2 -10185.123} C_VEL
LIN {X 0,Y 421.509,Z 328.56,A -85,B 0,C 180,E1 -10185.782,E2 -10185.782} C_VEL
LIN {X 0,Y 422.045,Z 319.767,A -85,B 0,C 180,E1 -10186.258,E2 -10186.258} C_VEL
LIN {X 0,Y 422.422,Z 309.837,A -85,B 0,C 180,E1 -10186.678,E2 -10186.678} C_VEL
LIN {X 0,Y 422.81,Z 299.984,A -85,B 0,C 180,E1 -10186.973,E2 -10186.973} C_VEL
LIN {X 0,Y 423.203,Z 275.273,A -85,B 0,C 180,E1 -10187.426,E2 -10187.426} C_VEL
LIN {X 0,Y 423.613,Z 218.029,A -85,B 0,C 180,E1 -10188.406,E2 -10188.406} C_VEL
LIN {X 0,Y 419.069,Z 192.689,A -85,B 0,C 180,E1 -10189.088,E2 -10189.088} C_VEL
LIN {X 0,Y 419.119,Z 191.389,A -85,B 0,C 180,E1 -10189.34,E2 -10189.34} C_VEL
LIN {X 0,Y 419.972,Z 178.615,A -85,B 0,C 180,E1 -10192.637,E2 -10192.637} C_VEL
LIN {X 0,Y 420.748,Z 168.723,A -85,B 0,C 180,E1 -10195.123,E2 -10195.123} C_VEL
LIN {X 0,Y 420.312,Z 164.221,A -85,B 0,C 180,E1 -10196.302,E2 -10196.302} C_VEL
LIN {X 0,Y 418.306,Z 153.996,A -85,B 0,C 180,E1 -10199.158,E2 -10199.158} C_VEL
LIN {X 0,Y 418.259,Z 153.883,A -85,B 0,C 180,E1 -10202.843,E2 -10202.843} C_VEL
LIN {X 0,Y 418.247,Z 153.881,A -85,B 0,C 180,E1 -10206.238,E2 -10206.238} C_VEL
LIN {X 0,Y 418.253,Z 153.87,A -85,B 0,C 180,E1 -10209.681,E2 -10209.681} C_VEL
LIN {X 0,Y 418.23,Z 153.886,A -85,B 0,C 180,E1 -10212.321,E2 -10212.321} C_VEL
LIN {X 0,Y 418.236,Z 153.884,A -85,B 0,C 180,E1 -10215.108,E2 -10215.108} C_VEL
LIN {X 0,Y 418.239,Z 153.888,A -85,B 0,C 180,E1 -10217.766,E2 -10217.766} C_VEL
LIN {X 0,Y 418.244,Z 153.877,A -85,B 0,C 180,E1 -10220.62,E2 -10220.62} C_VEL
LIN {X 0,Y 418.242,Z 153.881,A -85,B 0,C 180,E1 -10223.975,E2 -10223.975} C_VEL
LIN {X 0,Y 418.256,Z 153.877,A -85,B 0,C 180,E1 -10227.155,E2 -10227.155} C_VEL
LIN {X 0,Y 418.267,Z 153.882,A -85,B 0,C 180,E1 -10230.895,E2 -10230.895} C_VEL
LIN {X 0,Y 418.269,Z 153.87,A -85,B 0,C 180,E1 -10234.095,E2 -10234.095} C_VEL
LIN {X 0,Y 418.236,Z 153.886,A -85,B 0,C 180,E1 -10237.263,E2 -10237.263} C_VEL
LIN {X 0,Y 418.281,Z 153.868,A -85,B 0,C 180,E1 -10240.364,E2 -10240.364} C_VEL
LIN {X 0,Y 418.315,Z 153.87,A -85,B 0,C 180,E1 -10243.404,E2 -10243.404} C_VEL
LIN {X 0,Y 418.344,Z 153.869,A -85,B 0,C 180,E1 -10246.999,E2 -10246.999} C_VEL
LIN {X 0,Y 418.338,Z 153.853,A -85,B 0,C 180,E1 -10250.328,E2 -10250.328} C_VEL
LIN {X 0,Y 418.491,Z 153.851,A -85,B 0,C 180,E1 -10253.248,E2 -10253.248} C_VEL
LIN {X 0,Y 418.336,Z 153.873,A -85,B 0,C 180,E1 -10255.181,E2 -10255.181} C_VEL
LIN {X 0,Y 418.539,Z 153.843,A -85,B 0,C 180,E1 -10258.075,E2 -10258.075} C_VEL
LIN {X 0,Y 418.667,Z 153.812,A -85,B 0,C 180,E1 -10259.999,E2 -10259.999} C_VEL
LIN {X 0,Y 418.507,Z 153.849,A -85,B 0,C 180,E1 -10262.887,E2 -10262.887} C_VEL
LIN {X 0,Y 418.49,Z 153.85,A -85,B 0,C 180,E1 -10266.751,E2 -10266.751} C_VEL
LIN {X 0,Y 418.396,Z 153.849,A -85,B 0,C 180,E1 -10268.695,E2 -10268.695} C_VEL
LIN {X 0,Y 418.311,Z 153.864,A -85,B 0,C 180,E1 -10271.631,E2 -10271.631} C_VEL
LIN {X 0,Y 418.298,Z 153.878,A -85,B 0,C 180,E1 -10274.597,E2 -10274.597} C_VEL
LIN {X 0,Y 418.283,Z 153.872,A -85,B 0,C 180,E1 -10277.603,E2 -10277.603} C_VEL
LIN {X 0,Y 418.245,Z 153.876,A -85,B 0,C 180,E1 -10280.663,E2 -10280.663} C_VEL
LIN {X 0,Y 418.284,Z 153.884,A -85,B 0,C 180,E1 -10283.781,E2 -10283.781} C_VEL
LIN {X 0,Y 418.305,Z 153.864,A -85,B 0,C 180,E1 -10287.07,E2 -10287.07} C_VEL
LIN {X 0,Y 418.254,Z 153.884,A -85,B 0,C 180,E1 -10290.271,E2 -10290.271} C_VEL
LIN {X 0,Y 418.244,Z 153.875,A -85,B 0,C 180,E1 -10293.677,E2 -10293.677} C_VEL
LIN {X 0,Y 418.241,Z 153.888,A -85,B 0,C 180,E1 -10297.223,E2 -10297.223} C_VEL
LIN {X 0,Y 418.247,Z 153.878,A -85,B 0,C 180,E1 -10299.682,E2 -10299.682} C_VEL
LIN {X 0,Y 418.227,Z 153.884,A -85,B 0,C 180,E1 -10302.321,E2 -10302.321} C_VEL
LIN {X 0,Y 418.237,Z 153.881,A -85,B 0,C 180,E1 -10305.109,E2 -10305.109} C_VEL
LIN {X 0,Y 418.236,Z 153.853,A -85,B 0,C 180,E1 -10307.767,E2 -10307.767} C_VEL
LIN {X 0,Y 418.252,Z 153.886,A -85,B 0,C 180,E1 -10311.559,E2 -10311.559} C_VEL
LIN {X 0,Y 418.255,Z 153.865,A -85,B 0,C 180,E1 -10315.159,E2 -10315.159} C_VEL
LIN {X 0,Y 418.245,Z 153.886,A -85,B 0,C 180,E1 -10317.472,E2 -10317.472} C_VEL
LIN {X 0,Y 418.273,Z 153.871,A -85,B 0,C 180,E1 -10320.893,E2 -10320.893} C_VEL
LIN {X 0,Y 418.267,Z 153.885,A -85,B 0,C 180,E1 -10324.096,E2 -10324.096} C_VEL
LIN {X 0,Y 418.234,Z 153.889,A -85,B 0,C 180,E1 -10327.264,E2 -10327.264} C_VEL
LIN {X 0,Y 418.279,Z 153.885,A -85,B 0,C 180,E1 -10330.364,E2 -10330.364} C_VEL
LIN {X 0,Y 418.313,Z 153.879,A -85,B 0,C 180,E1 -10333.405,E2 -10333.405} C_VEL
LIN {X 0,Y 418.342,Z 153.876,A -85,B 0,C 180,E1 -10336.999,E2 -10336.999} C_VEL
LIN {X 0,Y 418.338,Z 153.878,A -85,B 0,C 180,E1 -10340.329,E2 -10340.329} C_VEL
LIN {X 0,Y 418.491,Z 153.857,A -85,B 0,C 180,E1 -10343.249,E2 -10343.249} C_VEL
LIN {X 0,Y 418.337,Z 153.877,A -85,B 0,C 180,E1 -10345.182,E2 -10345.182} C_VEL
LIN {X 0,Y 418.541,Z 153.852,A -85,B 0,C 180,E1 -10348.075,E2 -10348.075} C_VEL
LIN {X 0,Y 418.67,Z 153.837,A -85,B 0,C 180,E1 -10350,E2 -10350} C_VEL
LIN {X 0,Y 418.507,Z 153.855,A -85,B 0,C 180,E1 -10352.888,E2 -10352.888} C_VEL
LIN {X 0,Y 418.491,Z 153.857,A -85,B 0,C 180,E1 -10356.751,E2 -10356.751} C_VEL
LIN {X 0,Y 418.338,Z 153.878,A -85,B 0,C 180,E1 -10359.671,E2 -10359.671} C_VEL
LIN {X 0,Y 418.319,Z 153.879,A -85,B 0,C 180,E1 -10363.324,E2 -10363.324} C_VEL
LIN {X 0,Y 417.625,Z 153.967,A -85,B 0,C 180,E1 -10364.128,E2 -10364.128} C_VEL
LIN {X 0,Y 414.747,Z 154.325,A -85,B 0,C 180,E1 -10365.433,E2 -10365.433} C_VEL
LIN {X 0,Y 412.334,Z 154.624,A -85,B 0,C 180,E1 -10366.487,E2 -10366.487} C_VEL
LIN {X 0,Y 411.312,Z 154.753,A -85,B 0,C 180,E1 -10367.302,E2 -10367.302} C_VEL
LIN {X 0,Y 411.236,Z 154.76,A -85,B 0,C 180,E1 -10367.578,E2 -10367.578} C_VEL
LIN {X 0,Y 411.193,Z 154.767,A -85,B 0,C 180,E1 -10371.034,E2 -10371.034} C_VEL
LIN {X 0,Y 411.223,Z 154.761,A -85,B 0,C 180,E1 -10374.215,E2 -10374.215} C_VEL
LIN {X 0,Y 411.255,Z 154.757,A -85,B 0,C 180,E1 -10377.478,E2 -10377.478} C_VEL
LIN {X 0,Y 411.198,Z 154.76,A -85,B 0,C 180,E1 -10380.847,E2 -10380.847} C_VEL
LIN {X 0,Y 411.201,Z 154.744,A -85,B 0,C 180,E1 -10384.334,E2 -10384.334} C_VEL
LIN {X 0,Y 411.194,Z 154.764,A -85,B 0,C 180,E1 -10387.973,E2 -10387.973} C_VEL
LIN {X 0,Y 411.158,Z 154.738,A -85,B 0,C 180,E1 -10391.228,E2 -10391.228} C_VEL
LIN {X 0,Y 411.176,Z 154.755,A -85,B 0,C 180,E1 -10394.49,E2 -10394.49} C_VEL
LIN {X 0,Y 411.174,Z 154.765,A -85,B 0,C 180,E1 -10398.195,E2 -10398.195} C_VEL
LIN {X 0,Y 411.217,Z 154.76,A -85,B 0,C 180,E1 -10400.777,E2 -10400.777} C_VEL
LIN {X 0,Y 411.195,Z 154.756,A -85,B 0,C 180,E1 -10404.472,E2 -10404.472} C_VEL
LIN {X 0,Y 411.202,Z 154.761,A -85,B 0,C 180,E1 -10406.874,E2 -10406.874} C_VEL
LIN {X 0,Y 411.234,Z 154.754,A -85,B 0,C 180,E1 -10410.643,E2 -10410.643} C_VEL
LIN {X 0,Y 411.234,Z 154.745,A -85,B 0,C 180,E1 -10413.619,E2 -10413.619} C_VEL
LIN {X 0,Y 411.199,Z 154.762,A -85,B 0,C 180,E1 -10416.853,E2 -10416.853} C_VEL
LIN {X 0,Y 411.21,Z 154.746,A -85,B 0,C 180,E1 -10420.051,E2 -10420.051} C_VEL
LIN {X 0,Y 411.259,Z 154.748,A -85,B 0,C 180,E1 -10423.132,E2 -10423.132} C_VEL
LIN {X 0,Y 411.301,Z 154.746,A -85,B 0,C 180,E1 -10426.896,E2 -10426.896} C_VEL
LIN {X 0,Y 411.289,Z 154.731,A -85,B 0,C 180,E1 -10430.162,E2 -10430.162} C_VEL
LIN {X 0,Y 411.478,Z 154.721,A -85,B 0,C 180,E1 -10432.147,E2 -10432.147} C_VEL
LIN {X 0,Y 411.471,Z 154.73,A -85,B 0,C 180,E1 -10434.118,E2 -10434.118} C_VEL
LIN {X 0,Y 411.51,Z 154.71,A -85,B 0,C 180,E1 -10438.043,E2 -10438.043} C_VEL
LIN {X 0,Y 411.636,Z 154.687,A -85,B 0,C 180,E1 -10440.001,E2 -10440.001} C_VEL
LIN {X 0,Y 411.455,Z 154.725,A -85,B 0,C 180,E1 -10442.938,E2 -10442.938} C_VEL
LIN {X 0,Y 411.457,Z 154.727,A -85,B 0,C 180,E1 -10446.868,E2 -10446.868} C_VEL
LIN {X 0,Y 411.29,Z 154.73,A -85,B 0,C 180,E1 -10449.839,E2 -10449.839} C_VEL
LIN {X 0,Y 411.303,Z 154.747,A -85,B 0,C 180,E1 -10453.105,E2 -10453.105} C_VEL
LIN {X 0,Y 411.261,Z 154.748,A -85,B 0,C 180,E1 -10456.869,E2 -10456.869} C_VEL
LIN {X 0,Y 411.228,Z 154.746,A -85,B 0,C 180,E1 -10459.987,E2 -10459.987} C_VEL
LIN {X 0,Y 411.201,Z 154.764,A -85,B 0,C 180,E1 -10463.148,E2 -10463.148} C_VEL
LIN {X 0,Y 411.236,Z 154.746,A -85,B 0,C 180,E1 -10466.382,E2 -10466.382} C_VEL
LIN {X 0,Y 411.199,Z 154.761,A -85,B 0,C 180,E1 -10469.713,E2 -10469.713} C_VEL
LIN {X 0,Y 411.205,Z 154.752,A -85,B 0,C 180,E1 -10473.156,E2 -10473.156} C_VEL
LIN {X 0,Y 411.192,Z 154.764,A -85,B 0,C 180,E1 -10476.553,E2 -10476.553} C_VEL
LIN {X 0,Y 411.208,Z 154.754,A -85,B 0,C 180,E1 -10479.728,E2 -10479.728} C_VEL
LIN {X 0,Y 411.172,Z 154.765,A -85,B 0,C 180,E1 -10483.134,E2 -10483.134} C_VEL
LIN {X 0,Y 411.168,Z 154.766,A -85,B 0,C 180,E1 -10485.882,E2 -10485.882} C_VEL
LIN {X 0,Y 411.164,Z 154.754,A -85,B 0,C 180,E1 -10488.772,E2 -10488.772} C_VEL
LIN {X 0,Y 411.21,Z 154.761,A -85,B 0,C 180,E1 -10491.831,E2 -10491.831} C_VEL
LIN {X 0,Y 411.212,Z 154.755,A -85,B 0,C 180,E1 -10495.122,E2 -10495.122} C_VEL
LIN {X 0,Y 411.167,Z 154.762,A -85,B 0,C 180,E1 -10498.003,E2 -10498.003} C_VEL
LIN {X 0,Y 411.262,Z 154.907,A -85,B 0,C 180,E1 -10500.574,E2 -10500.574} C_VEL
LIN {X 0,Y 413.163,Z 164.736,A -85,B 0,C 180,E1 -10503.48,E2 -10503.48} C_VEL
LIN {X 0,Y 413.684,Z 169.936,A -85,B 0,C 180,E1 -10504.867,E2 -10504.867} C_VEL
LIN {X 0,Y 412.662,Z 184.422,A -85,B 0,C 180,E1 -10508.521,E2 -10508.521} C_VEL
LIN {X 0,Y 412.11,Z 192.227,A -85,B 0,C 180,E1 -10510.545,E2 -10510.545} C_VEL
LIN {X 0,Y 412.672,Z 195.62,A -85,B 0,C 180,E1 -10510.689,E2 -10510.689} C_VEL
LIN {X 0,Y 416.972,Z 219.69,A -85,B 0,C 180,E1 -10511.323,E2 -10511.323} C_VEL
LIN {X 0,Y 416.085,Z 297.129,A -85,B 0,C 180,E1 -10512.681,E2 -10512.681} C_VEL
LIN {X 0,Y 415.767,Z 307.024,A -85,B 0,C 180,E1 -10512.952,E2 -10512.952} C_VEL
LIN {X 0,Y 415.296,Z 316.998,A -85,B 0,C 180,E1 -10513.344,E2 -10513.344} C_VEL
LIN {X 0,Y 414.753,Z 327.362,A -85,B 0,C 180,E1 -10513.891,E2 -10513.891} C_VEL
LIN {X 0,Y 414.1,Z 336.494,A -85,B 0,C 180,E1 -10514.496,E2 -10514.496} C_VEL
LIN {X 0,Y 413.498,Z 345.492,A -85,B 0,C 180,E1 -10515.23,E2 -10515.23} C_VEL
LIN {X 0,Y 412.875,Z 353.993,A -85,B 0,C 180,E1 -10516.063,E2 -10516.063} C_VEL
LIN {X 0,Y 412.313,Z 361.617,A -85,B 0,C 180,E1 -10516.947,E2 -10516.947} C_VEL
LIN {X 0,Y 411.795,Z 368.838,A -85,B 0,C 180,E1 -10517.932,E2 -10517.932} C_VEL
LIN {X 0,Y 411.302,Z 375.04,A -85,B 0,C 180,E1 -10518.917,E2 -10518.917} C_VEL
LIN {X 0,Y 410.809,Z 381.577,A -85,B 0,C 180,E1 -10520.15,E2 -10520.15} C_VEL
LIN {X 0,Y 410.53,Z 386.079,A -85,B 0,C 180,E1 -10521.137,E2 -10521.137} C_VEL
LIN {X 0,Y 410.185,Z 391.569,A -85,B 0,C 180,E1 -10522.617,E2 -10522.617} C_VEL
LIN {X 0,Y 410.016,Z 395.893,A -85,B 0,C 180,E1 -10524.097,E2 -10524.097} C_VEL
LIN {X 0,Y 410.018,Z 398.26,A -85,B 0,C 180,E1 -10525.084,E2 -10525.084} C_VEL
LIN {X 0,Y 409.932,Z 400.056,A -85,B 0,C 180,E1 -10526.068,E2 -10526.068} C_VEL
LIN {X 0,Y 409.967,Z 402.501,A -85,B 0,C 180,E1 -10528.035,E2 -10528.035} C_VEL
LIN {X 0,Y 409.937,Z 403.088,A -85,B 0,C 180,E1 -10529.018,E2 -10529.018} C_VEL
LIN {X 0,Y 409.937,Z 403.088,A -85,B 0,C 180,E1 -10530.982,E2 -10530.982} C_VEL
LIN {X 0,Y 409.967,Z 402.501,A -85,B 0,C 180,E1 -10531.965,E2 -10531.965} C_VEL
LIN {X 0,Y 409.932,Z 400.056,A -85,B 0,C 180,E1 -10533.932,E2 -10533.932} C_VEL
LIN {X 0,Y 410.016,Z 397.11,A -85,B 0,C 180,E1 -10535.409,E2 -10535.409} C_VEL
LIN {X 0,Y 410.164,Z 393.124,A -85,B 0,C 180,E1 -10536.889,E2 -10536.889} C_VEL
LIN {X 0,Y 410.413,Z 387.995,A -85,B 0,C 180,E1 -10538.369,E2 -10538.369} C_VEL
LIN {X 0,Y 410.741,Z 382.733,A -85,B 0,C 180,E1 -10539.603,E2 -10539.603} C_VEL
LIN {X 0,Y 411.147,Z 376.415,A -85,B 0,C 180,E1 -10540.838,E2 -10540.838} C_VEL
LIN {X 0,Y 411.655,Z 370.465,A -85,B 0,C 180,E1 -10541.822,E2 -10541.822} C_VEL
LIN {X 0,Y 412.208,Z 363.538,A -85,B 0,C 180,E1 -10542.806,E2 -10542.806} C_VEL
LIN {X 0,Y 412.703,Z 356.491,A -85,B 0,C 180,E1 -10543.667,E2 -10543.667} C_VEL
LIN {X 0,Y 413.314,Z 348.167,A -85,B 0,C 180,E1 -10544.528,E2 -10544.528} C_VEL
LIN {X 0,Y 414.03,Z 338.127,A -85,B 0,C 180,E1 -10545.38,E2 -10545.38} C_VEL
LIN {X 0,Y 414.694,Z 328.369,A -85,B 0,C 180,E1 -10546.049,E2 -10546.049} C_VEL
LIN {X 0,Y 415.283,Z 318.288,A -85,B 0,C 180,E1 -10546.593,E2 -10546.593} C_VEL
LIN {X 0,Y 415.67,Z 308.772,A -85,B 0,C 180,E1 -10546.989,E2 -10546.989} C_VEL
LIN {X 0,Y 416.104,Z 298.463,A -85,B 0,C 180,E1 -10547.287,E2 -10547.287} C_VEL
LIN {X 0,Y 416.716,Z 245.583,A -85,B 0,C 180,E1 -10548.229,E2 -10548.229} C_VEL
LIN {X 0,Y 416.808,Z 218.62,A -85,B 0,C 180,E1 -10548.704,E2 -10548.704} C_VEL
LIN {X 0,Y 412.136,Z 192.5,A -85,B 0,C 180,E1 -10549.421,E2 -10549.421} C_VEL
LIN {X 0,Y 412.177,Z 191.199,A -85,B 0,C 180,E1 -10549.679,E2 -10549.679} C_VEL
LIN {X 0,Y 413.167,Z 177.475,A -85,B 0,C 180,E1 -10553.285,E2 -10553.285} C_VEL
LIN {X 0,Y 413.787,Z 169.001,A -85,B 0,C 180,E1 -10555.459,E2 -10555.459} C_VEL
LIN {X 0,Y 412.493,Z 161.048,A -85,B 0,C 180,E1 -10557.628,E2 -10557.628} C_VEL
LIN {X 0,Y 411.223,Z 154.78,A -85,B 0,C 180,E1 -10559.488,E2 -10559.488} C_VEL
LIN {X 0,Y 411.208,Z 154.762,A -85,B 0,C 180,E1 -10563.155,E2 -10563.155} C_VEL
LIN {X 0,Y 411.195,Z 154.762,A -85,B 0,C 180,E1 -10566.552,E2 -10566.552} C_VEL
LIN {X 0,Y 411.216,Z 154.746,A -85,B 0,C 180,E1 -10569.728,E2 -10569.728} C_VEL
LIN {X 0,Y 411.174,Z 154.767,A -85,B 0,C 180,E1 -10573.133,E2 -10573.133} C_VEL
LIN {X 0,Y 411.168,Z 154.767,A -85,B 0,C 180,E1 -10575.88,E2 -10575.88} C_VEL
LIN {X 0,Y 411.163,Z 154.766,A -85,B 0,C 180,E1 -10578.771,E2 -10578.771} C_VEL
LIN {X 0,Y 411.191,Z 154.764,A -85,B 0,C 180,E1 -10582.025,E2 -10582.025} C_VEL
LIN {X 0,Y 411.205,Z 154.75,A -85,B 0,C 180,E1 -10585.666,E2 -10585.666} C_VEL
LIN {X 0,Y 411.188,Z 154.768,A -85,B 0,C 180,E1 -10589.152,E2 -10589.152} C_VEL
LIN {X 0,Y 411.257,Z 154.743,A -85,B 0,C 180,E1 -10592.522,E2 -10592.522} C_VEL
LIN {X 0,Y 411.225,Z 154.756,A -85,B 0,C 180,E1 -10595.784,E2 -10595.784} C_VEL
LIN {X 0,Y 411.194,Z 154.757,A -85,B 0,C 180,E1 -10598.965,E2 -10598.965} C_VEL
LIN {X 0,Y 411.25,Z 154.737,A -85,B 0,C 180,E1 -10602.084,E2 -10602.084} C_VEL
LIN {X 0,Y 411.258,Z 154.755,A -85,B 0,C 180,E1 -10605.147,E2 -10605.147} C_VEL
LIN {X 0,Y 411.281,Z 154.747,A -85,B 0,C 180,E1 -10608.167,E2 -10608.167} C_VEL
LIN {X 0,Y 411.441,Z 154.719,A -85,B 0,C 180,E1 -10612.185,E2 -10612.185} C_VEL
LIN {X 0,Y 411.472,Z 154.727,A -85,B 0,C 180,E1 -10614.117,E2 -10614.117} C_VEL
LIN {X 0,Y 411.508,Z 154.718,A -85,B 0,C 180,E1 -10618.042,E2 -10618.042} C_VEL
LIN {X 0,Y 411.636,Z 154.687,A -85,B 0,C 180,E1 -10619.999,E2 -10619.999} C_VEL
LIN {X 0,Y 411.462,Z 154.726,A -85,B 0,C 180,E1 -10622.937,E2 -10622.937} C_VEL
LIN {X 0,Y 411.457,Z 154.725,A -85,B 0,C 180,E1 -10626.866,E2 -10626.866} C_VEL
LIN {X 0,Y 411.35,Z 154.725,A -85,B 0,C 180,E1 -10628.845,E2 -10628.845} C_VEL
LIN {X 0,Y 411.279,Z 154.742,A -85,B 0,C 180,E1 -10631.832,E2 -10631.832} C_VEL
LIN {X 0,Y 411.256,Z 154.754,A -85,B 0,C 180,E1 -10634.852,E2 -10634.852} C_VEL
LIN {X 0,Y 411.248,Z 154.742,A -85,B 0,C 180,E1 -10637.915,E2 -10637.915} C_VEL
LIN {X 0,Y 411.192,Z 154.755,A -85,B 0,C 180,E1 -10641.034,E2 -10641.034} C_VEL
LIN {X 0,Y 411.222,Z 154.758,A -85,B 0,C 180,E1 -10644.215,E2 -10644.215} C_VEL
LIN {X 0,Y 411.255,Z 154.741,A -85,B 0,C 180,E1 -10647.477,E2 -10647.477} C_VEL
LIN {X 0,Y 411.191,Z 154.763,A -85,B 0,C 180,E1 -10650.847,E2 -10650.847} C_VEL
LIN {X 0,Y 411.201,Z 154.747,A -85,B 0,C 180,E1 -10654.333,E2 -10654.333} C_VEL
LIN {X 0,Y 411.195,Z 154.764,A -85,B 0,C 180,E1 -10657.973,E2 -10657.973} C_VEL
LIN {X 0,Y 411.16,Z 154.761,A -85,B 0,C 180,E1 -10661.228,E2 -10661.228} C_VEL
LIN {X 0,Y 411.176,Z 154.764,A -85,B 0,C 180,E1 -10664.49,E2 -10664.49} C_VEL
LIN {X 0,Y 411.173,Z 154.732,A -85,B 0,C 180,E1 -10668.195,E2 -10668.195} C_VEL
LIN {X 0,Y 411.214,Z 154.757,A -85,B 0,C 180,E1 -10670.776,E2 -10670.776} C_VEL
LIN {X 0,Y 411.195,Z 154.75,A -85,B 0,C 180,E1 -10674.471,E2 -10674.471} C_VEL
LIN {X 0,Y 411.169,Z 154.767,A -85,B 0,C 180,E1 -10678.003,E2 -10678.003} C_VEL
LIN {X 0,Y 411.22,Z 154.752,A -85,B 0,C 180,E1 -10681.41,E2 -10681.41} C_VEL
LIN {X 0,Y 411.232,Z 154.763,A -85,B 0,C 180,E1 -10684.707,E2 -10684.707} C_VEL
LIN {X 0,Y 411.202,Z 154.765,A -85,B 0,C 180,E1 -10687.914,E2 -10687.914} C_VEL
LIN {X 0,Y 411.221,Z 154.763,A -85,B 0,C 180,E1 -10691.052,E2 -10691.052} C_VEL
LIN {X 0,Y 411.251,Z 154.76,A -85,B 0,C 180,E1 -10694.132,E2 -10694.132} C_VEL
LIN {X 0,Y 411.299,Z 154.753,A -85,B 0,C 180,E1 -10697.166,E2 -10697.166} C_VEL
LIN {X 0,Y 411.29,Z 154.755,A -85,B 0,C 180,E1 -10700.161,E2 -10700.161} C_VEL
LIN {X 0,Y 411.457,Z 154.734,A -85,B 0,C 180,E1 -10703.133,E2 -10703.133} C_VEL
LIN {X 0,Y 411.308,Z 154.753,A -85,B 0,C 180,E1 -10705.099,E2 -10705.099} C_VEL
LIN {X 0,Y 411.511,Z 154.728,A -85,B 0,C 180,E1 -10708.043,E2 -10708.043} C_VEL
LIN {X 0,Y 411.639,Z 154.713,A -85,B 0,C 180,E1 -10710,E2 -10710} C_VEL
LIN {X 0,Y 411.463,Z 154.733,A -85,B 0,C 180,E1 -10712.937,E2 -10712.937} C_VEL
LIN {X 0,Y 411.457,Z 154.734,A -85,B 0,C 180,E1 -10716.867,E2 -10716.867} C_VEL
LIN {X 0,Y 411.29,Z 154.755,A -85,B 0,C 180,E1 -10719.839,E2 -10719.839} C_VEL
LIN {X 0,Y 411.28,Z 154.755,A -85,B 0,C 180,E1 -10723.312,E2 -10723.312} C_VEL
LIN {X 0,Y 411.253,Z 154.759,A -85,B 0,C 180,E1 -10726.889,E2 -10726.889} C_VEL
LIN {X 0,Y 411.236,Z 154.76,A -85,B 0,C 180,E1 -10727.578,E2 -10727.578} C_VEL
LIN {X 0,Y 410.575,Z 154.845,A -85,B 0,C 180,E1 -10728.396,E2 -10728.396} C_VEL
LIN {X 0,Y 407.688,Z 155.206,A -85,B 0,C 180,E1 -10729.724,E2 -10729.724} C_VEL
LIN {X 0,Y 405.244,Z 155.509,A -85,B 0,C 180,E1 -10730.797,E2 -10730.797} C_VEL
LIN {X 0,Y 404.208,Z 155.638,A -85,B 0,C 180,E1 -10731.627,E2 -10731.627} C_VEL
LIN {X 0,Y 404.132,Z 155.644,A -85,B 0,C 180,E1 -10731.909,E2 -10731.909} C_VEL
LIN {X 0,Y 404.212,Z 155.637,A -85,B 0,C 180,E1 -10735.297,E2 -10735.297} C_VEL
LIN {X 0,Y 404.194,Z 155.633,A -85,B 0,C 180,E1 -10737.999,E2 -10737.999} C_VEL
LIN {X 0,Y 404.144,Z 155.645,A -85,B 0,C 180,E1 -10741.56,E2 -10741.56} C_VEL
LIN {X 0,Y 404.18,Z 155.618,A -85,B 0,C 180,E1 -10745.016,E2 -10745.016} C_VEL
LIN {X 0,Y 404.151,Z 155.643,A -85,B 0,C 180,E1 -10748.757,E2 -10748.757} C_VEL
LIN {X 0,Y 404.118,Z 155.611,A -85,B 0,C 180,E1 -10751.6,E2 -10751.6} C_VEL
LIN {X 0,Y 404.145,Z 155.63,A -85,B 0,C 180,E1 -10754.523,E2 -10754.523} C_VEL
LIN {X 0,Y 404.135,Z 155.642,A -85,B 0,C 180,E1 -10757.296,E2 -10757.296} C_VEL
LIN {X 0,Y 404.164,Z 155.629,A -85,B 0,C 180,E1 -10759.956,E2 -10759.956} C_VEL
LIN {X 0,Y 404.135,Z 155.642,A -85,B 0,C 180,E1 -10763.125,E2 -10763.125} C_VEL
LIN {X 0,Y 404.14,Z 155.629,A -85,B 0,C 180,E1 -10766.188,E2 -10766.188} C_VEL
LIN {X 0,Y 404.147,Z 155.641,A -85,B 0,C 180,E1 -10769.716,E2 -10769.716} C_VEL
LIN {X 0,Y 404.191,Z 155.621,A -85,B 0,C 180,E1 -10773.123,E2 -10773.123} C_VEL
LIN {X 0,Y 404.172,Z 155.635,A -85,B 0,C 180,E1 -10775.335,E2 -10775.335} C_VEL
LIN {X 0,Y 404.134,Z 155.636,A -85,B 0,C 180,E1 -10778.581,E2 -10778.581} C_VEL
LIN {X 0,Y 404.205,Z 155.614,A -85,B 0,C 180,E1 -10781.762,E2 -10781.762} C_VEL
LIN {X 0,Y 404.202,Z 155.633,A -85,B 0,C 180,E1 -10784.882,E2 -10784.882} C_VEL
LIN {X 0,Y 404.252,Z 155.619,A -85,B 0,C 180,E1 -10787.959,E2 -10787.959} C_VEL
LIN {X 0,Y 404.43,Z 155.598,A -85,B 0,C 180,E1 -10792.1,E2 -10792.1} C_VEL
LIN {X 0,Y 404.42,Z 155.61,A -85,B 0,C 180,E1 -10794.016,E2 -10794.016} C_VEL
LIN {X 0,Y 404.479,Z 155.586,A -85,B 0,C 180,E1 -10798.009,E2 -10798.009} C_VEL
LIN {X 0,Y 404.606,Z 155.562,A -85,B 0,C 180,E1 -10800.001,E2 -10800.001} C_VEL
LIN {X 0,Y 404.413,Z 155.603,A -85,B 0,C 180,E1 -10802.989,E2 -10802.989} C_VEL
LIN {X 0,Y 404.404,Z 155.607,A -85,B 0,C 180,E1 -10806.988,E2 -10806.988} C_VEL
LIN {X 0,Y 404.255,Z 155.606,A -85,B 0,C 180,E1 -10810.012,E2 -10810.012} C_VEL
LIN {X 0,Y 404.264,Z 155.625,A -85,B 0,C 180,E1 -10813.212,E2 -10813.212} C_VEL
LIN {X 0,Y 404.214,Z 155.622,A -85,B 0,C 180,E1 -10817.008,E2 -10817.008} C_VEL
LIN {X 0,Y 404.162,Z 155.626,A -85,B 0,C 180,E1 -10820.352,E2 -10820.352} C_VEL
LIN {X 0,Y 404.168,Z 155.636,A -85,B 0,C 180,E1 -10823.575,E2 -10823.575} C_VEL
LIN {X 0,Y 404.182,Z 155.624,A -85,B 0,C 180,E1 -10825.767,E2 -10825.767} C_VEL
LIN {X 0,Y 404.194,Z 155.623,A -85,B 0,C 180,E1 -10828,E2 -10828} C_VEL
LIN {X 0,Y 404.138,Z 155.64,A -85,B 0,C 180,E1 -10831.559,E2 -10831.559} C_VEL
LIN {X 0,Y 404.184,Z 155.629,A -85,B 0,C 180,E1 -10835.017,E2 -10835.017} C_VEL
LIN {X 0,Y 404.15,Z 155.638,A -85,B 0,C 180,E1 -10838.758,E2 -10838.758} C_VEL
LIN {X 0,Y 404.122,Z 155.642,A -85,B 0,C 180,E1 -10841.6,E2 -10841.6} C_VEL
LIN {X 0,Y 404.145,Z 155.638,A -85,B 0,C 180,E1 -10844.523,E2 -10844.523} C_VEL
LIN {X 0,Y 404.137,Z 155.642,A -85,B 0,C 180,E1 -10847.296,E2 -10847.296} C_VEL
LIN {X 0,Y 404.17,Z 155.621,A -85,B 0,C 180,E1 -10849.956,E2 -10849.956} C_VEL
LIN {X 0,Y 404.139,Z 155.641,A -85,B 0,C 180,E1 -10853.125,E2 -10853.125} C_VEL
LIN {X 0,Y 404.146,Z 155.646,A -85,B 0,C 180,E1 -10856.188,E2 -10856.188} C_VEL
LIN {X 0,Y 404.193,Z 155.633,A -85,B 0,C 180,E1 -10860.101,E2 -10860.101} C_VEL
LIN {X 0,Y 404.263,Z 155.951,A -85,B 0,C 180,E1 -10860.371,E2 -10860.371} C_VEL
LIN {X 0,Y 406.148,Z 165.592,A -85,B 0,C 180,E1 -10863.263,E2 -10863.263} C_VEL
LIN {X 0,Y 406.733,Z 170.804,A -85,B 0,C 180,E1 -10864.681,E2 -10864.681} C_VEL
LIN {X 0,Y 405.733,Z 184.234,A -85,B 0,C 180,E1 -10868.135,E2 -10868.135} C_VEL
LIN {X 0,Y 405.147,Z 192.065,A -85,B 0,C 180,E1 -10870.201,E2 -10870.201} C_VEL
LIN {X 0,Y 405.938,Z 196.307,A -85,B 0,C 180,E1 -10870.372,E2 -10870.372} C_VEL
LIN {X 0,Y 410.175,Z 220.189,A -85,B 0,C 180,E1 -10871.014,E2 -10871.014} C_VEL
LIN {X 0,Y 409.322,Z 296.938,A -85,B 0,C 180,E1 -10872.385,E2 -10872.385} C_VEL
LIN {X 0,Y 408.942,Z 307.706,A -85,B 0,C 180,E1 -10872.691,E2 -10872.691} C_VEL
LIN {X 0,Y 408.495,Z 316.807,A -85,B 0,C 180,E1 -10873.058,E2 -10873.058} C_VEL
LIN {X 0,Y 407.94,Z 327.17,A -85,B 0,C 180,E1 -10873.614,E2 -10873.614} C_VEL
LIN {X 0,Y 407.267,Z 336.302,A -85,B 0,C 180,E1 -10874.229,E2 -10874.229} C_VEL
LIN {X 0,Y 406.605,Z 345.299,A -85,B 0,C 180,E1 -10874.974,E2 -10874.974} C_VEL
LIN {X 0,Y 405.914,Z 353.937,A -85,B 0,C 180,E1 -10875.834,E2 -10875.834} C_VEL
LIN {X 0,Y 405.352,Z 361.424,A -85,B 0,C 180,E1 -10876.719,E2 -10876.719} C_VEL
LIN {X 0,Y 404.812,Z 368.646,A -85,B 0,C 180,E1 -10877.721,E2 -10877.721} C_VEL
LIN {X 0,Y 404.306,Z 374.848,A -85,B 0,C 180,E1 -10878.723,E2 -10878.723} C_VEL
LIN {X 0,Y 403.801,Z 381.385,A -85,B 0,C 180,E1 -10879.977,E2 -10879.977} C_VEL
LIN {X 0,Y 403.487,Z 385.887,A -85,B 0,C 180,E1 -10880.981,E2 -10880.981} C_VEL
LIN {X 0,Y 403.133,Z 391.377,A -85,B 0,C 180,E1 -10882.487,E2 -10882.487} C_VEL
LIN {X 0,Y 402.94,Z 395.701,A -85,B 0,C 180,E1 -10883.993,E2 -10883.993} C_VEL
LIN {X 0,Y 402.93,Z 398.068,A -85,B 0,C 180,E1 -10884.997,E2 -10884.997} C_VEL
LIN {X 0,Y 402.853,Z 399.865,A -85,B 0,C 180,E1 -10885.999,E2 -10885.999} C_VEL
LIN {X 0,Y 402.865,Z 402.309,A -85,B 0,C 180,E1 -10888.001,E2 -10888.001} C_VEL
LIN {X 0,Y 402.864,Z 402.897,A -85,B 0,C 180,E1 -10889,E2 -10889} C_VEL
LIN {X 0,Y 402.864,Z 402.897,A -85,B 0,C 180,E1 -10891,E2 -10891} C_VEL
LIN {X 0,Y 402.865,Z 402.309,A -85,B 0,C 180,E1 -10891.999,E2 -10891.999} C_VEL
LIN {X 0,Y 402.853,Z 399.865,A -85,B 0,C 180,E1 -10894.001,E2 -10894.001} C_VEL
LIN {X 0,Y 402.914,Z 396.918,A -85,B 0,C 180,E1 -10895.505,E2 -10895.505} C_VEL
LIN {X 0,Y 403.076,Z 392.931,A -85,B 0,C 180,E1 -10897.01,E2 -10897.01} C_VEL
LIN {X 0,Y 403.356,Z 387.802,A -85,B 0,C 180,E1 -10898.517,E2 -10898.517} C_VEL
LIN {X 0,Y 403.702,Z 382.54,A -85,B 0,C 180,E1 -10899.772,E2 -10899.772} C_VEL
LIN {X 0,Y 404.145,Z 376.222,A -85,B 0,C 180,E1 -10901.028,E2 -10901.028} C_VEL
LIN {X 0,Y 404.679,Z 370.273,A -85,B 0,C 180,E1 -10902.029,E2 -10902.029} C_VEL
LIN {X 0,Y 405.249,Z 363.345,A -85,B 0,C 180,E1 -10903.029,E2 -10903.029} C_VEL
LIN {X 0,Y 405.855,Z 355.164,A -85,B 0,C 180,E1 -10904.03,E2 -10904.03} C_VEL
LIN {X 0,Y 406.488,Z 346.786,A -85,B 0,C 180,E1 -10904.89,E2 -10904.89} C_VEL
LIN {X 0,Y 407.158,Z 337.935,A -85,B 0,C 180,E1 -10905.647,E2 -10905.647} C_VEL
LIN {X 0,Y 407.877,Z 328.177,A -85,B 0,C 180,E1 -10906.324,E2 -10906.324} C_VEL
LIN {X 0,Y 408.421,Z 319.384,A -85,B 0,C 180,E1 -10906.816,E2 -10906.816} C_VEL
LIN {X 0,Y 408.853,Z 309.455,A -85,B 0,C 180,E1 -10907.248,E2 -10907.248} C_VEL
LIN {X 0,Y 409.27,Z 299.602,A -85,B 0,C 180,E1 -10907.553,E2 -10907.553} C_VEL
LIN {X 0,Y 409.691,Z 275.053,A -85,B 0,C 180,E1 -10908.017,E2 -10908.017} C_VEL
LIN {X 0,Y 410.062,Z 219.493,A -85,B 0,C 180,E1 -10909.004,E2 -10909.004} C_VEL
LIN {X 0,Y 405.213,Z 192.287,A -85,B 0,C 180,E1 -10909.769,E2 -10909.769} C_VEL
LIN {X 0,Y 405.305,Z 190.061,A -85,B 0,C 180,E1 -10910.291,E2 -10910.291} C_VEL
LIN {X 0,Y 406.395,Z 176.248,A -85,B 0,C 180,E1 -10913.978,E2 -10913.978} C_VEL
LIN {X 0,Y 406.831,Z 170.103,A -85,B 0,C 180,E1 -10915.586,E2 -10915.586} C_VEL
LIN {X 0,Y 405.435,Z 161.823,A -85,B 0,C 180,E1 -10917.906,E2 -10917.906} C_VEL
LIN {X 0,Y 404.209,Z 155.651,A -85,B 0,C 180,E1 -10919.777,E2 -10919.777} C_VEL
LIN {X 0,Y 404.172,Z 155.64,A -85,B 0,C 180,E1 -10923.419,E2 -10923.419} C_VEL
LIN {X 0,Y 404.144,Z 155.636,A -85,B 0,C 180,E1 -10926.246,E2 -10926.246} C_VEL
LIN {X 0,Y 404.159,Z 155.637,A -85,B 0,C 180,E1 -10928.756,E2 -10928.756} C_VEL
LIN {X 0,Y 404.123,Z 155.634,A -85,B 0,C 180,E1 -10931.599,E2 -10931.599} C_VEL
LIN {X 0,Y 404.145,Z 155.639,A -85,B 0,C 180,E1 -10934.521,E2 -10934.521} C_VEL
LIN {X 0,Y 404.136,Z 155.646,A -85,B 0,C 180,E1 -10937.295,E2 -10937.295} C_VEL
LIN {X 0,Y 404.169,Z 155.631,A -85,B 0,C 180,E1 -10939.955,E2 -10939.955} C_VEL
LIN {X 0,Y 404.135,Z 155.646,A -85,B 0,C 180,E1 -10943.125,E2 -10943.125} C_VEL
LIN {X 0,Y 404.144,Z 155.628,A -85,B 0,C 180,E1 -10946.187,E2 -10946.187} C_VEL
LIN {X 0,Y 404.144,Z 155.641,A -85,B 0,C 180,E1 -10949.714,E2 -10949.714} C_VEL
LIN {X 0,Y 404.193,Z 155.62,A -85,B 0,C 180,E1 -10953.122,E2 -10953.122} C_VEL
LIN {X 0,Y 404.176,Z 155.637,A -85,B 0,C 180,E1 -10955.334,E2 -10955.334} C_VEL
LIN {X 0,Y 404.158,Z 155.639,A -85,B 0,C 180,E1 -10958.581,E2 -10958.581} C_VEL
LIN {X 0,Y 404.208,Z 155.613,A -85,B 0,C 180,E1 -10961.761,E2 -10961.761} C_VEL
LIN {X 0,Y 404.204,Z 155.635,A -85,B 0,C 180,E1 -10964.881,E2 -10964.881} C_VEL
LIN {X 0,Y 404.253,Z 155.621,A -85,B 0,C 180,E1 -10967.958,E2 -10967.958} C_VEL
LIN {X 0,Y 404.403,Z 155.595,A -85,B 0,C 180,E1 -10972.127,E2 -10972.127} C_VEL
LIN {X 0,Y 404.421,Z 155.604,A -85,B 0,C 180,E1 -10974.014,E2 -10974.014} C_VEL
LIN {X 0,Y 404.477,Z 155.594,A -85,B 0,C 180,E1 -10978.008,E2 -10978.008} C_VEL
LIN {X 0,Y 404.606,Z 155.562,A -85,B 0,C 180,E1 -10979.999,E2 -10979.999} C_VEL
LIN {X 0,Y 404.419,Z 155.603,A -85,B 0,C 180,E1 -10982.988,E2 -10982.988} C_VEL
LIN {X 0,Y 404.408,Z 155.602,A -85,B 0,C 180,E1 -10986.987,E2 -10986.987} C_VEL
LIN {X 0,Y 404.254,Z 155.606,A -85,B 0,C 180,E1 -10990.011,E2 -10990.011} C_VEL
LIN {X 0,Y 404.262,Z 155.623,A -85,B 0,C 180,E1 -10993.211,E2 -10993.211} C_VEL
LIN {X 0,Y 404.211,Z 155.626,A -85,B 0,C 180,E1 -10997.007,E2 -10997.007} C_VEL
LIN {X 0,Y 404.159,Z 155.63,A -85,B 0,C 180,E1 -11000.351,E2 -11000.351} C_VEL
LIN {X 0,Y 404.165,Z 155.642,A -85,B 0,C 180,E1 -11003.574,E2 -11003.574} C_VEL
LIN {X 0,Y 404.179,Z 155.629,A -85,B 0,C 180,E1 -11005.766,E2 -11005.766} C_VEL
LIN {X 0,Y 404.192,Z 155.624,A -85,B 0,C 180,E1 -11007.999,E2 -11007.999} C_VEL
LIN {X 0,Y 404.137,Z 155.646,A -85,B 0,C 180,E1 -11011.558,E2 -11011.558} C_VEL
LIN {X 0,Y 404.18,Z 155.623,A -85,B 0,C 180,E1 -11015.016,E2 -11015.016} C_VEL
LIN {X 0,Y 404.153,Z 155.641,A -85,B 0,C 180,E1 -11018.756,E2 -11018.756} C_VEL
LIN {X 0,Y 404.119,Z 155.641,A -85,B 0,C 180,E1 -11021.6,E2 -11021.6} C_VEL
LIN {X 0,Y 404.145,Z 155.64,A -85,B 0,C 180,E1 -11024.523,E2 -11024.523} C_VEL
LIN {X 0,Y 404.133,Z 155.61,A -85,B 0,C 180,E1 -11027.296,E2 -11027.296} C_VEL
LIN {X 0,Y 404.164,Z 155.631,A -85,B 0,C 180,E1 -11029.955,E2 -11029.955} C_VEL
LIN {X 0,Y 404.135,Z 155.64,A -85,B 0,C 180,E1 -11033.124,E2 -11033.124} C_VEL
LIN {X 0,Y 404.141,Z 155.627,A -85,B 0,C 180,E1 -11036.188,E2 -11036.188} C_VEL
LIN {X 0,Y 404.152,Z 155.634,A -85,B 0,C 180,E1 -11039.716,E2 -11039.716} C_VEL
LIN {X 0,Y 404.191,Z 155.639,A -85,B 0,C 180,E1 -11043.123,E2 -11043.123} C_VEL
LIN {X 0,Y 404.173,Z 155.64,A -85,B 0,C 180,E1 -11045.334,E2 -11045.334} C_VEL
LIN {X 0,Y 404.135,Z 155.647,A -85,B 0,C 180,E1 -11048.581,E2 -11048.581} C_VEL
LIN {X 0,Y 404.206,Z 155.637,A -85,B 0,C 180,E1 -11051.762,E2 -11051.762} C_VEL
LIN {X 0,Y 404.202,Z 155.638,A -85,B 0,C 180,E1 -11054.882,E2 -11054.882} C_VEL
LIN {X 0,Y 404.253,Z 155.632,A -85,B 0,C 180,E1 -11057.959,E2 -11057.959} C_VEL
LIN {X 0,Y 404.43,Z 155.611,A -85,B 0,C 180,E1 -11062.1,E2 -11062.1} C_VEL
LIN {X 0,Y 404.421,Z 155.611,A -85,B 0,C 180,E1 -11064.015,E2 -11064.015} C_VEL
LIN {X 0,Y 404.479,Z 155.603,A -85,B 0,C 180,E1 -11068.009,E2 -11068.009} C_VEL
LIN {X 0,Y 404.608,Z 155.588,A -85,B 0,C 180,E1 -11070,E2 -11070} C_VEL
LIN {X 0,Y 404.42,Z 155.611,A -85,B 0,C 180,E1 -11072.988,E2 -11072.988} C_VEL
LIN {X 0,Y 404.408,Z 155.613,A -85,B 0,C 180,E1 -11076.987,E2 -11076.987} C_VEL
LIN {X 0,Y 404.255,Z 155.632,A -85,B 0,C 180,E1 -11080.012,E2 -11080.012} C_VEL
LIN {X 0,Y 404.262,Z 155.631,A -85,B 0,C 180,E1 -11083.211,E2 -11083.211} C_VEL
LIN {X 0,Y 404.212,Z 155.637,A -85,B 0,C 180,E1 -11087.007,E2 -11087.007} C_VEL
LIN {X 0,Y 404.16,Z 155.642,A -85,B 0,C 180,E1 -11090.352,E2 -11090.352} C_VEL
LIN {X 0,Y 404.132,Z 155.644,A -85,B 0,C 180,E1 -11091.909,E2 -11091.909} C_VEL
LIN {X 0,Y 403.489,Z 155.726,A -85,B 0,C 180,E1 -11092.74,E2 -11092.74} C_VEL
LIN {X 0,Y 400.657,Z 156.08,A -85,B 0,C 180,E1 -11094.092,E2 -11094.092} C_VEL
LIN {X 0,Y 398.248,Z 156.381,A -85,B 0,C 180,E1 -11095.184,E2 -11095.184} C_VEL
LIN {X 0,Y 397.214,Z 156.508,A -85,B 0,C 180,E1 -11096.028,E2 -11096.028} C_VEL
LIN {X 0,Y 397.13,Z 156.516,A -85,B 0,C 180,E1 -11096.314,E2 -11096.314} C_VEL
LIN {X 0,Y 397.122,Z 156.507,A -85,B 0,C 180,E1 -11098.543,E2 -11098.543} C_VEL
LIN {X 0,Y 397.108,Z 156.519,A -85,B 0,C 180,E1 -11102.069,E2 -11102.069} C_VEL
LIN {X 0,Y 397.115,Z 156.501,A -85,B 0,C 180,E1 -11105.504,E2 -11105.504} C_VEL
LIN {X 0,Y 397.126,Z 156.516,A -85,B 0,C 180,E1 -11108.862,E2 -11108.862} C_VEL
LIN {X 0,Y 397.064,Z 156.487,A -85,B 0,C 180,E1 -11112.267,E2 -11112.267} C_VEL
LIN {X 0,Y 397.087,Z 156.517,A -85,B 0,C 180,E1 -11115.068,E2 -11115.068} C_VEL
LIN {X 0,Y 397.063,Z 156.522,A -85,B 0,C 180,E1 -11118.021,E2 -11118.021} C_VEL
LIN {X 0,Y 397.128,Z 156.517,A -85,B 0,C 180,E1 -11121.138,E2 -11121.138} C_VEL
LIN {X 0,Y 397.115,Z 156.508,A -85,B 0,C 180,E1 -11124.497,E2 -11124.497} C_VEL
LIN {X 0,Y 397.075,Z 156.52,A -85,B 0,C 180,E1 -11127.929,E2 -11127.929} C_VEL
LIN {X 0,Y 397.12,Z 156.507,A -85,B 0,C 180,E1 -11131.457,E2 -11131.457} C_VEL
LIN {X 0,Y 397.148,Z 156.508,A -85,B 0,C 180,E1 -11134.488,E2 -11134.488} C_VEL
LIN {X 0,Y 397.105,Z 156.517,A -85,B 0,C 180,E1 -11137.086,E2 -11137.086} C_VEL
LIN {X 0,Y 397.143,Z 156.493,A -85,B 0,C 180,E1 -11140.353,E2 -11140.353} C_VEL
LIN {X 0,Y 397.162,Z 156.505,A -85,B 0,C 180,E1 -11143.554,E2 -11143.554} C_VEL
LIN {X 0,Y 397.224,Z 156.5,A -85,B 0,C 180,E1 -11146.703,E2 -11146.703} C_VEL
LIN {X 0,Y 397.214,Z 156.483,A -85,B 0,C 180,E1 -11149.809,E2 -11149.809} C_VEL
LIN {X 0,Y 397.36,Z 156.48,A -85,B 0,C 180,E1 -11152.889,E2 -11152.889} C_VEL
LIN {X 0,Y 397.252,Z 156.499,A -85,B 0,C 180,E1 -11154.926,E2 -11154.926} C_VEL
LIN {X 0,Y 397.448,Z 156.462,A -85,B 0,C 180,E1 -11157.974,E2 -11157.974} C_VEL
LIN {X 0,Y 397.575,Z 156.436,A -85,B 0,C 180,E1 -11160.001,E2 -11160.001} C_VEL
LIN {X 0,Y 397.373,Z 156.48,A -85,B 0,C 180,E1 -11163.042,E2 -11163.042} C_VEL
LIN {X 0,Y 397.372,Z 156.481,A -85,B 0,C 180,E1 -11166.092,E2 -11166.092} C_VEL
LIN {X 0,Y 397.25,Z 156.478,A -85,B 0,C 180,E1 -11169.162,E2 -11169.162} C_VEL
LIN {X 0,Y 397.216,Z 156.497,A -85,B 0,C 180,E1 -11172.259,E2 -11172.259} C_VEL
LIN {X 0,Y 397.177,Z 156.507,A -85,B 0,C 180,E1 -11175.393,E2 -11175.393} C_VEL
LIN {X 0,Y 397.16,Z 156.49,A -85,B 0,C 180,E1 -11178.574,E2 -11178.574} C_VEL
LIN {X 0,Y 397.107,Z 156.515,A -85,B 0,C 180,E1 -11181.818,E2 -11181.818} C_VEL
LIN {X 0,Y 397.151,Z 156.501,A -85,B 0,C 180,E1 -11185.513,E2 -11185.513} C_VEL
LIN {X 0,Y 397.12,Z 156.507,A -85,B 0,C 180,E1 -11188.544,E2 -11188.544} C_VEL
LIN {X 0,Y 397.077,Z 156.52,A -85,B 0,C 180,E1 -11192.072,E2 -11192.072} C_VEL
LIN {X 0,Y 397.118,Z 156.511,A -85,B 0,C 180,E1 -11195.504,E2 -11195.504} C_VEL
LIN {X 0,Y 397.126,Z 156.511,A -85,B 0,C 180,E1 -11198.861,E2 -11198.861} C_VEL
LIN {X 0,Y 397.068,Z 156.525,A -85,B 0,C 180,E1 -11202.268,E2 -11202.268} C_VEL
LIN {X 0,Y 397.087,Z 156.519,A -85,B 0,C 180,E1 -11205.069,E2 -11205.069} C_VEL
LIN {X 0,Y 397.067,Z 156.519,A -85,B 0,C 180,E1 -11208.022,E2 -11208.022} C_VEL
LIN {X 0,Y 397.133,Z 156.511,A -85,B 0,C 180,E1 -11211.139,E2 -11211.139} C_VEL
LIN {X 0,Y 397.121,Z 156.506,A -85,B 0,C 180,E1 -11214.497,E2 -11214.497} C_VEL
LIN {X 0,Y 397.08,Z 156.516,A -85,B 0,C 180,E1 -11217.929,E2 -11217.929} C_VEL
LIN {X 0,Y 397.173,Z 156.658,A -85,B 0,C 180,E1 -11220.014,E2 -11220.014} C_VEL
LIN {X 0,Y 399.292,Z 167.504,A -85,B 0,C 180,E1 -11223.332,E2 -11223.332} C_VEL
LIN {X 0,Y 399.736,Z 172.71,A -85,B 0,C 180,E1 -11224.764,E2 -11224.764} C_VEL
LIN {X 0,Y 398.68,Z 186,A -85,B 0,C 180,E1 -11228.273,E2 -11228.273} C_VEL
LIN {X 0,Y 398.225,Z 191.863,A -85,B 0,C 180,E1 -11229.841,E2 -11229.841} C_VEL
LIN {X 0,Y 398.891,Z 195.643,A -85,B 0,C 180,E1 -11230.002,E2 -11230.002} C_VEL
LIN {X 0,Y 403.498,Z 221.232,A -85,B 0,C 180,E1 -11230.71,E2 -11230.71} C_VEL
LIN {X 0,Y 402.57,Z 296.747,A -85,B 0,C 180,E1 -11232.08,E2 -11232.08} C_VEL
LIN {X 0,Y 402.18,Z 307.515,A -85,B 0,C 180,E1 -11232.39,E2 -11232.39} C_VEL
LIN {X 0,Y 401.719,Z 316.615,A -85,B 0,C 180,E1 -11232.764,E2 -11232.764} C_VEL
LIN {X 0,Y 401.142,Z 326.979,A -85,B 0,C 180,E1 -11233.328,E2 -11233.328} C_VEL
LIN {X 0,Y 400.421,Z 336.11,A -85,B 0,C 180,E1 -11233.953,E2 -11233.953} C_VEL
LIN {X 0,Y 399.734,Z 345.107,A -85,B 0,C 180,E1 -11234.709,E2 -11234.709} C_VEL
LIN {X 0,Y 399.104,Z 352.705,A -85,B 0,C 180,E1 -11235.468,E2 -11235.468} C_VEL
LIN {X 0,Y 398.404,Z 361.394,A -85,B 0,C 180,E1 -11236.505,E2 -11236.505} C_VEL
LIN {X 0,Y 397.851,Z 368.453,A -85,B 0,C 180,E1 -11237.503,E2 -11237.503} C_VEL
LIN {X 0,Y 397.288,Z 374.654,A -85,B 0,C 180,E1 -11238.521,E2 -11238.521} C_VEL
LIN {X 0,Y 396.781,Z 381.192,A -85,B 0,C 180,E1 -11239.798,E2 -11239.798} C_VEL
LIN {X 0,Y 396.42,Z 385.693,A -85,B 0,C 180,E1 -11240.819,E2 -11240.819} C_VEL
LIN {X 0,Y 396.062,Z 391.185,A -85,B 0,C 180,E1 -11242.352,E2 -11242.352} C_VEL
LIN {X 0,Y 395.863,Z 395.509,A -85,B 0,C 180,E1 -11243.885,E2 -11243.885} C_VEL
LIN {X 0,Y 395.843,Z 397.876,A -85,B 0,C 180,E1 -11244.907,E2 -11244.907} C_VEL
LIN {X 0,Y 395.775,Z 399.673,A -85,B 0,C 180,E1 -11245.927,E2 -11245.927} C_VEL
LIN {X 0,Y 395.763,Z 402.117,A -85,B 0,C 180,E1 -11247.965,E2 -11247.965} C_VEL
LIN {X 0,Y 395.792,Z 402.706,A -85,B 0,C 180,E1 -11248.983,E2 -11248.983} C_VEL
LIN {X 0,Y 395.792,Z 402.706,A -85,B 0,C 180,E1 -11251.017,E2 -11251.017} C_VEL
LIN {X 0,Y 395.763,Z 402.117,A -85,B 0,C 180,E1 -11252.035,E2 -11252.035} C_VEL
LIN {X 0,Y 395.775,Z 399.673,A -85,B 0,C 180,E1 -11254.073,E2 -11254.073} C_VEL
LIN {X 0,Y 395.843,Z 397.876,A -85,B 0,C 180,E1 -11255.093,E2 -11255.093} C_VEL
LIN {X 0,Y 395.92,Z 394.27,A -85,B 0,C 180,E1 -11256.625,E2 -11256.625} C_VEL
LIN {X 0,Y 396.178,Z 389.525,A -85,B 0,C 180,E1 -11258.159,E2 -11258.159} C_VEL
LIN {X 0,Y 396.603,Z 383.504,A -85,B 0,C 180,E1 -11259.691,E2 -11259.691} C_VEL
LIN {X 0,Y 397.03,Z 377.406,A -85,B 0,C 180,E1 -11260.97,E2 -11260.97} C_VEL
LIN {X 0,Y 397.705,Z 370.08,A -85,B 0,C 180,E1 -11262.243,E2 -11262.243} C_VEL
LIN {X 0,Y 398.29,Z 363.152,A -85,B 0,C 180,E1 -11263.261,E2 -11263.261} C_VEL
LIN {X 0,Y 398.954,Z 354.971,A -85,B 0,C 180,E1 -11264.278,E2 -11264.278} C_VEL
LIN {X 0,Y 399.603,Z 346.594,A -85,B 0,C 180,E1 -11265.153,E2 -11265.153} C_VEL
LIN {X 0,Y 400.302,Z 337.742,A -85,B 0,C 180,E1 -11265.922,E2 -11265.922} C_VEL
LIN {X 0,Y 401.06,Z 327.986,A -85,B 0,C 180,E1 -11266.61,E2 -11266.61} C_VEL
LIN {X 0,Y 401.633,Z 319.192,A -85,B 0,C 180,E1 -11267.109,E2 -11267.109} C_VEL
LIN {X 0,Y 402.09,Z 309.263,A -85,B 0,C 180,E1 -11267.548,E2 -11267.548} C_VEL
LIN {X 0,Y 402.516,Z 299.41,A -85,B 0,C 180,E1 -11267.857,E2 -11267.857} C_VEL
LIN {X 0,Y 402.954,Z 274.938,A -85,B 0,C 180,E1 -11268.327,E2 -11268.327} C_VEL
LIN {X 0,Y 403.357,Z 220.397,A -85,B 0,C 180,E1 -11269.312,E2 -11269.312} C_VEL
LIN {X 0,Y 398.299,Z 192.332,A -85,B 0,C 180,E1 -11270.109,E2 -11270.109} C_VEL
LIN {X 0,Y 398.25,Z 191.318,A -85,B 0,C 180,E1 -11270.263,E2 -11270.263} C_VEL
LIN {X 0,Y 399.452,Z 177.075,A -85,B 0,C 180,E1 -11274.146,E2 -11274.146} C_VEL
LIN {X 0,Y 399.844,Z 170.96,A -85,B 0,C 180,E1 -11275.787,E2 -11275.787} C_VEL
LIN {X 0,Y 398.417,Z 162.847,A -85,B 0,C 180,E1 -11278.116,E2 -11278.116} C_VEL
LIN {X 0,Y 397.138,Z 156.534,A -85,B 0,C 180,E1 -11280.056,E2 -11280.056} C_VEL
LIN {X 0,Y 397.12,Z 156.522,A -85,B 0,C 180,E1 -11283.717,E2 -11283.717} C_VEL
LIN {X 0,Y 397.097,Z 156.519,A -85,B 0,C 180,E1 -11287.209,E2 -11287.209} C_VEL
LIN {X 0,Y 397.102,Z 156.5,A -85,B 0,C 180,E1 -11290.445,E2 -11290.445} C_VEL
LIN {X 0,Y 397.101,Z 156.523,A -85,B 0,C 180,E1 -11293.648,E2 -11293.648} C_VEL
LIN {X 0,Y 397.102,Z 156.518,A -85,B 0,C 180,E1 -11296.52,E2 -11296.52} C_VEL
LIN {X 0,Y 397.112,Z 156.509,A -85,B 0,C 180,E1 -11300.422,E2 -11300.422} C_VEL
LIN {X 0,Y 397.107,Z 156.513,A -85,B 0,C 180,E1 -11304.265,E2 -11304.265} C_VEL
LIN {X 0,Y 397.113,Z 156.505,A -85,B 0,C 180,E1 -11306.726,E2 -11306.726} C_VEL
LIN {X 0,Y 397.123,Z 156.514,A -85,B 0,C 180,E1 -11310.295,E2 -11310.295} C_VEL
LIN {X 0,Y 397.193,Z 156.493,A -85,B 0,C 180,E1 -11312.609,E2 -11312.609} C_VEL
LIN {X 0,Y 397.131,Z 156.511,A -85,B 0,C 180,E1 -11315.981,E2 -11315.981} C_VEL
LIN {X 0,Y 397.137,Z 156.501,A -85,B 0,C 180,E1 -11319.704,E2 -11319.704} C_VEL
LIN {X 0,Y 397.18,Z 156.495,A -85,B 0,C 180,E1 -11322.844,E2 -11322.844} C_VEL
LIN {X 0,Y 397.226,Z 156.503,A -85,B 0,C 180,E1 -11326.702,E2 -11326.702} C_VEL
LIN {X 0,Y 397.215,Z 156.483,A -85,B 0,C 180,E1 -11329.808,E2 -11329.808} C_VEL
LIN {X 0,Y 397.353,Z 156.483,A -85,B 0,C 180,E1 -11332.887,E2 -11332.887} C_VEL
LIN {X 0,Y 397.252,Z 156.501,A -85,B 0,C 180,E1 -11334.925,E2 -11334.925} C_VEL
LIN {X 0,Y 397.446,Z 156.47,A -85,B 0,C 180,E1 -11337.973,E2 -11337.973} C_VEL
LIN {X 0,Y 397.575,Z 156.436,A -85,B 0,C 180,E1 -11339.999,E2 -11339.999} C_VEL
LIN {X 0,Y 397.378,Z 156.48,A -85,B 0,C 180,E1 -11343.041,E2 -11343.041} C_VEL
LIN {X 0,Y 397.36,Z 156.48,A -85,B 0,C 180,E1 -11347.111,E2 -11347.111} C_VEL
LIN {X 0,Y 397.214,Z 156.483,A -85,B 0,C 180,E1 -11350.191,E2 -11350.191} C_VEL
LIN {X 0,Y 397.222,Z 156.5,A -85,B 0,C 180,E1 -11353.321,E2 -11353.321} C_VEL
LIN {X 0,Y 397.177,Z 156.502,A -85,B 0,C 180,E1 -11357.155,E2 -11357.155} C_VEL
LIN {X 0,Y 397.098,Z 156.51,A -85,B 0,C 180,E1 -11360.73,E2 -11360.73} C_VEL
LIN {X 0,Y 397.128,Z 156.516,A -85,B 0,C 180,E1 -11364.018,E2 -11364.018} C_VEL
LIN {X 0,Y 397.19,Z 156.492,A -85,B 0,C 180,E1 -11367.39,E2 -11367.39} C_VEL
LIN {X 0,Y 397.078,Z 156.522,A -85,B 0,C 180,E1 -11370.882,E2 -11370.882} C_VEL
LIN {X 0,Y 397.121,Z 156.5,A -85,B 0,C 180,E1 -11374.493,E2 -11374.493} C_VEL
LIN {X 0,Y 397.101,Z 156.518,A -85,B 0,C 180,E1 -11378.274,E2 -11378.274} C_VEL
LIN {X 0,Y 397.084,Z 156.511,A -85,B 0,C 180,E1 -11380.908,E2 -11380.908} C_VEL
LIN {X 0,Y 397.099,Z 156.52,A -85,B 0,C 180,E1 -11383.648,E2 -11383.648} C_VEL
LIN {X 0,Y 397.1,Z 156.497,A -85,B 0,C 180,E1 -11386.52,E2 -11386.52} C_VEL
LIN {X 0,Y 397.109,Z 156.511,A -85,B 0,C 180,E1 -11390.423,E2 -11390.423} C_VEL
LIN {X 0,Y 397.104,Z 156.506,A -85,B 0,C 180,E1 -11394.265,E2 -11394.265} C_VEL
LIN {X 0,Y 397.111,Z 156.507,A -85,B 0,C 180,E1 -11396.727,E2 -11396.727} C_VEL
LIN {X 0,Y 397.13,Z 156.503,A -85,B 0,C 180,E1 -11400.297,E2 -11400.297} C_VEL
LIN {X 0,Y 397.191,Z 156.51,A -85,B 0,C 180,E1 -11402.61,E2 -11402.61} C_VEL
LIN {X 0,Y 397.129,Z 156.518,A -85,B 0,C 180,E1 -11405.982,E2 -11405.982} C_VEL
LIN {X 0,Y 397.135,Z 156.518,A -85,B 0,C 180,E1 -11409.705,E2 -11409.705} C_VEL
LIN {X 0,Y 397.178,Z 156.514,A -85,B 0,C 180,E1 -11412.845,E2 -11412.845} C_VEL
LIN {X 0,Y 397.225,Z 156.508,A -85,B 0,C 180,E1 -11416.703,E2 -11416.703} C_VEL
LIN {X 0,Y 397.215,Z 156.509,A -85,B 0,C 180,E1 -11419.809,E2 -11419.809} C_VEL
LIN {X 0,Y 397.361,Z 156.491,A -85,B 0,C 180,E1 -11422.888,E2 -11422.888} C_VEL
LIN {X 0,Y 397.252,Z 156.504,A -85,B 0,C 180,E1 -11424.925,E2 -11424.925} C_VEL
LIN {X 0,Y 397.46,Z 156.769,A -85,B 0,C 180,E1 -11428.227,E2 -11428.227} C_VEL
LIN {X 0,Y 397.651,Z 156.873,A -85,B 0,C 180,E1 -11430,E2 -11430} C_VEL
LIN {X 0,Y 397.378,Z 156.565,A -85,B 0,C 180,E1 -11433.041,E2 -11433.041} C_VEL
LIN {X 0,Y 397.361,Z 156.491,A -85,B 0,C 180,E1 -11437.112,E2 -11437.112} C_VEL
LIN {X 0,Y 397.215,Z 156.509,A -85,B 0,C 180,E1 -11440.191,E2 -11440.191} C_VEL
LIN {X 0,Y 397.223,Z 156.508,A -85,B 0,C 180,E1 -11443.321,E2 -11443.321} C_VEL
LIN {X 0,Y 397.178,Z 156.513,A -85,B 0,C 180,E1 -11447.155,E2 -11447.155} C_VEL
LIN {X 0,Y 397.099,Z 156.522,A -85,B 0,C 180,E1 -11450.73,E2 -11450.73} C_VEL
LIN {X 0,Y 397.129,Z 156.518,A -85,B 0,C 180,E1 -11454.018,E2 -11454.018} C_VEL
LIN {X 0,Y 397.13,Z 156.516,A -85,B 0,C 180,E1 -11456.314,E2 -11456.314} C_VEL
LIN {X 0,Y 396.459,Z 156.603,A -85,B 0,C 180,E1 -11457.161,E2 -11457.161} C_VEL
LIN {X 0,Y 393.584,Z 156.948,A -85,B 0,C 180,E1 -11458.537,E2 -11458.537} C_VEL
LIN {X 0,Y 391.15,Z 157.251,A -85,B 0,C 180,E1 -11459.648,E2 -11459.648} C_VEL
LIN {X 0,Y 390.106,Z 157.384,A -85,B 0,C 180,E1 -11460.508,E2 -11460.508} C_VEL
LIN {X 0,Y 390.022,Z 157.396,A -85,B 0,C 180,E1 -11460.799,E2 -11460.799} C_VEL
LIN {X 0,Y 390.063,Z 157.376,A -85,B 0,C 180,E1 -11464.025,E2 -11464.025} C_VEL
